(* CODESYS project UralKoksWin.project

Project tree, tasks and I/O mapping:
  Device : SPK1xx[M01], Production association OWEN, order no. 4, version 3.5.11.54
    application Application
      libraries: Standard, * (System); Util, * (System)
      task MainTask (cyclic, interval t#20ms, priority 1) calls PLC_PRG, MECH
      task VISU_TASK (cyclic, interval 100 ms, priority 31) calls VisuElems.Visu_Prg, CountWebCli
      task Task_Chain (cyclic, interval t#20ms, priority 1) calls Chain
      task TrendRecordingTask (cyclic, interval 100 ms, priority 31) calls VisuTrendStorageAccess.GlobalInstances.g_TrendRecordingManager.CyclicCall
      program PLC_PRG [LD]
      visualisation VFrADiag
      data type MV210_202
      data type MU210_402
      data type TRM201
      data type Vector75
      visualisation VFr4Baraban
      visualisation VMain
      visualisation VFr1Main
      image pool ImagePool
      visualisation VFr2KonvFrak
      visualisation VFr3Grohot
      visualisation VFr5Gorelka
      visualisation VFr6Dedusting
      text list TextList
      data type Vector100
      data type ABB330
      global variables GVL
      program MECH [CFC]
      data type PME
      data type VLT2800
      program Chain [ST]
      text list STEPS
      function block Motor [LD]
      program CountWebCli [ST]
      visualisation VFr7RandE
    Info : Info, Production association OWEN, version 3.5.11.5002
        unmapped channels: VENDOR, DEVICE, SERIAL, RUNTIME, FIRMWARE, LINUX, TARGET, PROJECT, AUTHOR, VERSION, PROFILE, LASTCHANGES
    Screen : Screen, Production association OWEN, version 3.5.11.5001
        unmapped channels: Get Brightness, Dim time, Off time, Full brightness, Dim brightness, Off brightness, Dim visu name, Off visu name, On visu name, Wake up
    Debug : Debug, Production association OWEN, version 3.5.11.5001
        unmapped channels: RAM used, RAM free, Open files, Processor usage, Core temp, Enable Debug, Debug pause
    OwenRTC : OwenRTC, Production association OWEN, version 3.5.11.5001
        unmapped channels: Year, Month, Day, Hour, Minute, Second, Day of Week, Week of Year, Format Date, Format Time, UTC Offset, NTP Enabled, NTP Error, System Timer, New Year, New Month, New Day, New Hour, New Minute, New Second, New UTC Offset, Set Settings DT, Enable NTP, Prefer Server
    OwenCloud : OwenCloud, Production association OWEN, version 3.5.11.5001
        unmapped channels: OwenCloud enabled, Enable OwenCloud, Token
    Drives : Drives, Production association OWEN, version 3.5.11.5001
        unmapped channels: FS size, FS used, FS free, USB Mounted, USB Unmount done, USB size, USB used, USB free, MMC Mounted, MMC Unmount done, MMC size, MMC used, MMC free, Enable Drives, USB Unmount, MMC Unmount
    Network : Network, Production association OWEN, version 3.5.11.5001
        unmapped channels: DHCP enabled, IP, Mask, Gateway, MAC, Hostname, Enable DHCP, New IP, New Mask, New Gateway, New Hostname, Set Settings
    Watchdog : Watchdog, Production association OWEN, version 3.5.11.5001
        unmapped channels: Exception Handling, Last Exception Code, Last Exception Description, Last Exception Time, Hardware Watchdog Flag, Reboot
    Buzzer : Buzzer, Production association OWEN, version 3.5.11.5001
        unmapped channels: Buzzer enabled, Enable Buzzer
    Ethernet : Ethernet, 3S - Smart Software Solutions GmbH, version 3.5.11.0
        settings: IPAddress = [192,168,1,151]; SubnetMask = [255,255,255,0]; GatewayAddress = [0,0,0,0]; MACAddress = [16#E4,16#1E,16#0A,16#00,16#16,16#C1]; NetworkInterfaceName = 'eth0'; NetworkInterfaceName = "eth0"; SaveCommunicationSettings = FALSE
      Modbus_TCP_Master : Modbus TCP Master, 3S - Smart Software Solutions GmbH, version 3.5.11.30
          settings: AutoReconnect = TRUE
        MU210_402DO : Modbus TCP Slave, 3S - Smart Software Solutions GmbH, version 3.5.11.30
            settings: Unit-ID = 1; IPAddress = [192, 168, 1, 153]; DO.Function Code = 16; DO.Read Offset = 0; DO.Read Length = 0; DO.Write Offset = 16#01D6; DO.Write Length = 1; DO.Cycle Time = 20
            output Application.MECH.K40.xMODBUS_Run : BOOL  // DO.DO.Bit0
            output Application.MECH.K25.xMODBUS_Run : BOOL  // DO.DO.Bit1
            output Application.MECH.K10.xMODBUS_Run : BOOL  // DO.DO.Bit2
            output Application.MECH.K0.xOUT_Run : BOOL  // DO.DO.Bit3
            output Application.MECH.Gr.xOUT_Run : BOOL  // DO.DO.Bit4
            output Application.MECH.PD.xMODBUS_Run : BOOL  // DO.DO.Bit5
            output Application.MECH.BR.xOUT_Run : BOOL  // DO.DO.Bit6
            output Application.MECH.Ded.xOUT_MODBUS_Run : BOOL  // DO.DO.Bit7
            output Application.MECH.EL.xOUT_MODBUS_Run : BOOL  // DO.DO.Bit8
            output Application.MECH.xGorRun : BOOL  // DO.DO.Bit9
            output Application.MECH.xVibRun : BOOL  // DO.DO.Bit10
            output Application.PLC_PRG.DOutput1.xDO12 : BOOL  // DO.DO.Bit11
            output Application.MECH.xGorAck : BOOL  // DO.DO.Bit12
            output Application.Chain.xLampPUSK : BOOL  // DO.DO.Bit13
            output Application.MECH.xDrob_OUT_Run : BOOL  // DO.DO.Bit14
            output Application.PLC_PRG.DOutput1.xDO16 : BOOL  // DO.DO.Bit15
            unmapped channels: DO
        MV210_202DI : Modbus TCP Slave, 3S - Smart Software Solutions GmbH, version 3.5.11.30
            settings: Unit-ID = 1; IPAddress = [192, 168, 1, 152]; DI.Function Code = 3; DI.Read Offset = 16#0033; DI.Read Length = 2; DI.Write Offset = 0; DI.Write Length = 0; DI.Cycle Time = 20
            input  Application.PLC_PRG.DInput1.xDI1 : BOOL  // DI.DI.Bit0
            input  Application.PLC_PRG.DInput1.xDI2 : BOOL  // DI.DI.Bit1
            input  Application.PLC_PRG.DInput1.xDI3 : BOOL  // DI.DI.Bit2
            input  Application.PLC_PRG.DInput1.xDI4 : BOOL  // DI.DI.Bit3
            input  Application.PLC_PRG.DInput1.xDI5 : BOOL  // DI.DI.Bit4
            input  Application.PLC_PRG.DInput1.xDI6 : BOOL  // DI.DI.Bit5
            input  Application.PLC_PRG.DInput1.xDI7 : BOOL  // DI.DI.Bit6
            input  Application.PLC_PRG.DInput1.xDI8 : BOOL  // DI.DI.Bit7
            input  Application.PLC_PRG.DInput1.xDI9 : BOOL  // DI.DI.Bit8
            input  Application.PLC_PRG.DInput1.xDI10 : BOOL  // DI.DI.Bit9
            input  Application.PLC_PRG.DInput1.xDI11 : BOOL  // DI.DI.Bit10
            input  Application.PLC_PRG.DInput1.xDI12 : BOOL  // DI.DI.Bit11
            input  Application.PLC_PRG.DInput1.xDI13 : BOOL  // DI.DI.Bit12
            input  Application.PLC_PRG.DInput1.xDI14 : BOOL  // DI.DI.Bit13
            input  Application.PLC_PRG.DInput1.xDI15 : BOOL  // DI.DI.Bit14
            input  Application.PLC_PRG.DInput1.xDI16 : BOOL  // DI.DI.Bit15
            input  Application.PLC_PRG.DInput1.xDI17 : BOOL  // DI.DI.Bit0
            input  Application.PLC_PRG.DInput1.xDI18 : BOOL  // DI.DI.Bit1
            input  Application.PLC_PRG.DInput1.xDI19 : BOOL  // DI.DI.Bit2
            input  Application.PLC_PRG.DInput1.xDI20 : BOOL  // DI.DI.Bit3
            unmapped channels: DI
        MV210_202DI2 : Modbus TCP Slave, 3S - Smart Software Solutions GmbH, version 3.5.11.30
            settings: Unit-ID = 1; IPAddress = [192, 168, 1, 154]; DI.Function Code = 3; DI.Read Offset = 16#0033; DI.Read Length = 2; DI.Write Offset = 0; DI.Write Length = 0; DI.Cycle Time = 20
            input  Application.PLC_PRG.DInput2.xDI1 : BOOL  // DI.DI.Bit0
            input  Application.PLC_PRG.DInput2.xDI2 : BOOL  // DI.DI.Bit1
            input  Application.MECH.xGorFault : BOOL  // DI.DI.Bit2
            input  Application.MECH.xGorWork : BOOL  // DI.DI.Bit3
            input  Application.MECH.xGor2Stup : BOOL  // DI.DI.Bit4
            input  Application.PLC_PRG.DInput2.xDI6 : BOOL  // DI.DI.Bit5
            input  Application.PLC_PRG.DInput2.xDI7 : BOOL  // DI.DI.Bit6
            input  Application.PLC_PRG.DInput2.xDI8 : BOOL  // DI.DI.Bit7
            input  Application.PLC_PRG.DInput2.xDI9 : BOOL  // DI.DI.Bit8
            input  Application.PLC_PRG.DInput2.xDI10 : BOOL  // DI.DI.Bit9
            input  Application.PLC_PRG.DInput2.xDI11 : BOOL  // DI.DI.Bit10
            input  Application.PLC_PRG.DInput2.xDI12 : BOOL  // DI.DI.Bit11
            input  Application.PLC_PRG.DInput2.xDI13 : BOOL  // DI.DI.Bit12
            input  Application.PLC_PRG.DInput2.xDI14 : BOOL  // DI.DI.Bit13
            input  Application.PLC_PRG.DInput2.xDI15 : BOOL  // DI.DI.Bit14
            input  Application.PLC_PRG.DInput2.xDI16 : BOOL  // DI.DI.Bit15
            input  Application.PLC_PRG.DInput2.xDI17 : BOOL  // DI.DI.Bit0
            input  Application.PLC_PRG.DInput2.xDI18 : BOOL  // DI.DI.Bit1
            input  Application.PLC_PRG.DInput2.xDI19 : BOOL  // DI.DI.Bit2
            input  Application.PLC_PRG.DInput2.xDI20 : BOOL  // DI.DI.Bit3
            unmapped channels: DI
    COM2 : Modbus COM, 3S - Smart Software Solutions GmbH, version 3.5.11.20
        settings: DataBits = 8; StopBits = 2; ComPort = 2
      Master_2 : Modbus Master, COM Port, 3S - Smart Software Solutions GmbH, version 3.5.11.20
          settings: Transmission = 'RTU'; ResponseTimeout = 1000; TimeBetweenFrames = 20; Auto-restart communication = TRUE
        DedustingSlave : Modbus Slave, COM Port, 3S - Smart Software Solutions GmbH, version 3.5.10.30
            settings: SlaveAddress = 30; ResponseTimeout = 1000; UseExtendedFunctionCodes = TRUE; Current.Function Code = 3; Current.Read Offset = 16#1004; Current.Read Length = 1; Current.Write Offset = 0; Current.Write Length = 0; Current.Cycle Time = 1000; PVSpeed.Function Code = 3; PVSpeed.Read Offset = 16#1001; PVSpeed.Read Length = 1; PVSpeed.Write Offset = 0; PVSpeed.Write Length = 0; PVSpeed.Cycle Time = 1000; SPSpeed.Function Code = 6; SPSpeed.Read Offset = 0; SPSpeed.Read Length = 0; SPSpeed.Write Offset = 16#1000; SPSpeed.Write Length = 1; SPSpeed.Cycle Time = 1000
            input  Application.MECH.Ded.iIN_MODBUS_Iengie : WORD  // Current.Current
            input  Application.MECH.Ded.iIN_MODBUS_PVSpeed : WORD  // PVSpeed.PVSpeed
            output Application.MECH.Ded.iOUT_MODBUS_SPSpeed : WORD  // SPSpeed.SPSpeed
            unmapped channels: Current, PVSpeed, SPSpeed
        ElevatorSlave : Modbus Slave, COM Port, 3S - Smart Software Solutions GmbH, version 3.5.10.30
            settings: SlaveAddress = 25; ResponseTimeout = 1000; UseExtendedFunctionCodes = TRUE; PVSpeed.Function Code = 3; PVSpeed.Read Offset = 16#1001; PVSpeed.Read Length = 1; PVSpeed.Write Offset = 0; PVSpeed.Write Length = 0; PVSpeed.Cycle Time = 1000; Current.Function Code = 3; Current.Read Offset = 16#1004; Current.Read Length = 1; Current.Write Offset = 0; Current.Write Length = 0; Current.Cycle Time = 1000; SPspeed.Function Code = 6; SPspeed.Read Offset = 0; SPspeed.Read Length = 0; SPspeed.Write Offset = 16#1000; SPspeed.Write Length = 1; SPspeed.Cycle Time = 1000
            input  Application.MECH.EL.iIN_MODBUS_PVSpeed : WORD  // PVSpeed.PVSpeed
            input  Application.MECH.EL.iIN_MODBUS_Iengie : WORD  // Current.Current
            output Application.MECH.EL.iOUT_MODBUS_SPSpeed : WORD  // SPspeed.SPspeed
            unmapped channels: PVSpeed, Current, SPspeed
        VentilatorSlave : Modbus Slave, COM Port, 3S - Smart Software Solutions GmbH, version 3.5.10.30
            settings: SlaveAddress = 35; ResponseTimeout = 1000; UseExtendedFunctionCodes = TRUE; PVSpeed.Function Code = 3; PVSpeed.Read Offset = 16#1001; PVSpeed.Read Length = 1; PVSpeed.Write Offset = 0; PVSpeed.Write Length = 0; PVSpeed.Cycle Time = 1000; StatWord.Function Code = 3; StatWord.Read Offset = 16#3000; StatWord.Read Length = 1; StatWord.Write Offset = 0; StatWord.Write Length = 0; StatWord.Cycle Time = 1000; BR_Speed.Function Code = 3; BR_Speed.Read Offset = 16#100B; BR_Speed.Read Length = 1; BR_Speed.Write Offset = 0; BR_Speed.Write Length = 0; BR_Speed.Cycle Time = 100
            input  Application.MECH.iInMBVentPVSpeed : WORD  // PVSpeed.PVSpeed
            input  Application.MECH.xVentWorkBit1 : BOOL  // StatWord.StatWord.Bit0
            input  Application.MECH.xVentWorkBit2 : BOOL  // StatWord.StatWord.Bit1
            input  Application.MECH.BR.iIN_MODBUS_PVSpeed : WORD  // BR_Speed.BR_Speed
            unmapped channels: PVSpeed, StatWord, BR_Speed
    COM1 : Modbus COM, 3S - Smart Software Solutions GmbH, version 3.5.11.20
        settings: DataBits = 8; StopBits = 2; ComPort = 1
      Master_1 : Modbus Master, COM Port, 3S - Smart Software Solutions GmbH, version 3.5.11.20
          settings: Transmission = 'RTU'; ResponseTimeout = 1000; TimeBetweenFrames = 10; Auto-restart communication = TRUE
        Konv40Slave : Modbus Slave, COM Port, 3S - Smart Software Solutions GmbH, version 3.5.10.30
            settings: SlaveAddress = 5; ResponseTimeout = 1000; UseExtendedFunctionCodes = TRUE; SPSpeed.Function Code = 6; SPSpeed.Read Offset = 0; SPSpeed.Read Length = 0; SPSpeed.Write Offset = 16#1000; SPSpeed.Write Length = 1; SPSpeed.Cycle Time = 1000; PVSpeed.Function Code = 3; PVSpeed.Read Offset = 16#1001; PVSpeed.Read Length = 1; PVSpeed.Write Offset = 0; PVSpeed.Write Length = 0; PVSpeed.Cycle Time = 1000; Current.Function Code = 3; Current.Read Offset = 16#1004; Current.Read Length = 1; Current.Write Offset = 0; Current.Write Length = 0; Current.Cycle Time = 1000; MI.Function Code = 3; MI.Read Offset = 16#1008; MI.Read Length = 1; MI.Write Offset = 0; MI.Write Length = 0; MI.Cycle Time = 1000
            output Application.MECH.K40.iMODBUS_SPSpeed : WORD  // SPSpeed.SPSpeed
            input  Application.MECH.K40.iMODBUS_PVSpeed : WORD  // PVSpeed.PVSpeed
            input  Application.MECH.K40.iMODBUS_Iengie : WORD  // Current.Current
            input  Application.MECH.KM_K0 : BOOL  // MI.MI.Bit3
            input  Application.MECH.KM_Gr : BOOL  // MI.MI.Bit4
            unmapped channels: SPSpeed, PVSpeed, Current, MI
        PodachaSlave : Modbus Slave, COM Port, 3S - Smart Software Solutions GmbH, version 3.5.10.30
            settings: SlaveAddress = 20; ResponseTimeout = 1000; UseExtendedFunctionCodes = TRUE; PVSpeed.Function Code = 3; PVSpeed.Read Offset = 16#0004; PVSpeed.Read Length = 3; PVSpeed.Write Offset = 0; PVSpeed.Write Length = 0; PVSpeed.Cycle Time = 1000
            input  Application.MECH.PD.iMODBUS_SPSpeed : WORD  // PVSpeed.PVSpeed
            input  Application.MECH.PD.iMODBUS_PVSpeed : WORD  // PVSpeed.PVSpeed
            input  Application.MECH.PD.iMODBUS_Iengie : WORD  // PVSpeed.PVSpeed
            unmapped channels: PVSpeed
        Konv25Slave : Modbus Slave, COM Port, 3S - Smart Software Solutions GmbH, version 3.5.10.30
            settings: SlaveAddress = 10; ResponseTimeout = 1000; UseExtendedFunctionCodes = TRUE; SPSpeed.Function Code = 6; SPSpeed.Read Offset = 0; SPSpeed.Read Length = 0; SPSpeed.Write Offset = 16#1000; SPSpeed.Write Length = 1; SPSpeed.Cycle Time = 1000; PVSpeed.Function Code = 3; PVSpeed.Read Offset = 16#1001; PVSpeed.Read Length = 1; PVSpeed.Write Offset = 0; PVSpeed.Write Length = 0; PVSpeed.Cycle Time = 1000; Current.Function Code = 3; Current.Read Offset = 16#1004; Current.Read Length = 1; Current.Write Offset = 0; Current.Write Length = 0; Current.Cycle Time = 1000
            output Application.MECH.K25.iMODBUS_SPSpeed : WORD  // SPSpeed.SPSpeed
            input  Application.MECH.K25.iMODBUS_PVSpeed : WORD  // PVSpeed.PVSpeed
            input  Application.MECH.K25.iMODBUS_Iengie : WORD  // Current.Current
            unmapped channels: SPSpeed, PVSpeed, Current
        Konv10Slave : Modbus Slave, COM Port, 3S - Smart Software Solutions GmbH, version 3.5.10.30
            settings: SlaveAddress = 15; ResponseTimeout = 1000; UseExtendedFunctionCodes = TRUE; SPSpeed.Function Code = 6; SPSpeed.Read Offset = 0; SPSpeed.Read Length = 0; SPSpeed.Write Offset = 16#1000; SPSpeed.Write Length = 1; SPSpeed.Cycle Time = 1000; PVSpeed.Function Code = 3; PVSpeed.Read Offset = 16#1001; PVSpeed.Read Length = 1; PVSpeed.Write Offset = 0; PVSpeed.Write Length = 0; PVSpeed.Cycle Time = 1000; Current.Function Code = 3; Current.Read Offset = 16#1004; Current.Read Length = 1; Current.Write Offset = 0; Current.Write Length = 0; Current.Cycle Time = 1000
            output Application.MECH.K10.iMODBUS_SPSpeed : WORD  // SPSpeed.SPSpeed
            input  Application.MECH.K10.iMODBUS_PVSpeed : WORD  // PVSpeed.PVSpeed
            input  Application.MECH.K10.iMODBUS_Iengie : WORD  // Current.Current
            unmapped channels: SPSpeed, PVSpeed, Current
    COM3 : Modbus COM, 3S - Smart Software Solutions GmbH, version 3.5.11.20
        settings: DataBits = 8; StopBits = 2; ComPort = 3
      Master_3 : Modbus Master, COM Port, 3S - Smart Software Solutions GmbH, version 3.5.11.20
          settings: Transmission = 'RTU'; ResponseTimeout = 1000; TimeBetweenFrames = 10; Auto-restart communication = TRUE
        TRMGorelkaSlave : Modbus Slave, COM Port, 3S - Smart Software Solutions GmbH, version 3.5.10.30
            settings: SlaveAddress = 40; ResponseTimeout = 1000; UseExtendedFunctionCodes = TRUE; PV_SP.Function Code = 3; PV_SP.Read Offset = 16#0001; PV_SP.Read Length = 1; PV_SP.Write Offset = 0; PV_SP.Write Length = 0; PV_SP.Cycle Time = 1000; temp_SP.Function Code = 3; temp_SP.Read Offset = 16#0002; temp_SP.Read Length = 1; temp_SP.Write Offset = 0; temp_SP.Write Length = 0; temp_SP.Cycle Time = 1000; STAT.Function Code = 3; STAT.Read Offset = 16#0000; STAT.Read Length = 1; STAT.Write Offset = 0; STAT.Write Length = 0; STAT.Cycle Time = 1000
            input  Application.MECH.iInMBGorPVTemp : WORD  // PV_SP.PV_SP
            input  Application.MECH.iInMBGorSPTemp : WORD  // temp_SP.temp_SP
            input  Application.MECH.xGorNagrevONOFF : BOOL  // STAT.STAT.Bit4
            unmapped channels: PV_SP, temp_SP, STAT
        TRMDedustingSlave : Modbus Slave, COM Port, 3S - Smart Software Solutions GmbH, version 3.5.10.30
            settings: SlaveAddress = 45; ResponseTimeout = 1000; UseExtendedFunctionCodes = TRUE; PV_SP.Function Code = 3; PV_SP.Read Offset = 16#0001; PV_SP.Read Length = 1; PV_SP.Write Offset = 0; PV_SP.Write Length = 0; PV_SP.Cycle Time = 1000
            input  Application.MECH.iInMBDedPVTemp : WORD  // PV_SP.PV_SP
            unmapped channels: PV_SP
  text list GlobalTextList
  5ce3da45-db07-42e7-a21c-a00fff4ed8f6|img\fonFrame.png
  text list System
  5ce3da45-db07-42e7-a21c-a00fff4ed8f6|img\frame1.png
  5ce3da45-db07-42e7-a21c-a00fff4ed8f6|img\333.png
*)

// Device/Application/MV210_202
TYPE MV210_202 :
STRUCT
	xDI1: BOOL;
	xDI2: BOOL;
	xDI3: BOOL;
	xDI4: BOOL;
	xDI5: BOOL;
	xDI6: BOOL;
	xDI7: BOOL;
	xDI8: BOOL;
	xDI9: BOOL;
	xDI10: BOOL;
	xDI11: BOOL;
	xDI12: BOOL;
	xDI13: BOOL;
	xDI14: BOOL;
	xDI15: BOOL;
	xDI16: BOOL;
	xDI17: BOOL;
	xDI18: BOOL;
	xDI19: BOOL;
	xDI20: BOOL;
END_STRUCT
END_TYPE

// Device/Application/MU210_402
TYPE MU210_402 :
STRUCT
	xDO1: BOOL;
	xDO2: BOOL;
	xDO3: BOOL;
	xDO4: BOOL;
	xDO5: BOOL;
	xDO6: BOOL;
	xDO7: BOOL;
	xDO8: BOOL;
	xDO9: BOOL;
	xDO10: BOOL;
	xDO11: BOOL;
	xDO12: BOOL;
	xDO13: BOOL;
	xDO14: BOOL;
	xDO15: BOOL;
	xDO16: BOOL;
END_STRUCT
END_TYPE

// Device/Application/TRM201
TYPE TRM201 :
STRUCT
	iPV: INT;
	iSP: INT;
	nagrevONOFF: BOOL;
	
END_STRUCT
END_TYPE

// Device/Application/Vector75
TYPE Vector75 :
STRUCT
	iOUT_MODBUS_SPSpeed,
	iIN_MODBUS_PVSpeed,
	iIN_MODBUS_Iengie: INT;
	

	xIN_Run: BOOL;
	xOUT_MODBUS_Run:BOOL;
	xOUT_Ready: BOOL;
	xOUT_Error: BOOL;
	xOUT_Work: BOOL;

	xIN_Error: BOOL;

	iOUT_PVRotation: INT;
	iOUT_PVSpeed: INT; 

	rOUT_Current: REAL;
	
	iIN_MODBUS_AI: INT;
END_STRUCT
END_TYPE

// Device/Application/Vector100
TYPE Vector100 :
STRUCT
	iMODBUS_SPSpeed,
	iMODBUS_PVSpeed,
	iMODBUS_Iengie: INT;
	

	xIN_Run: BOOL;
	xMODBUS_Run:BOOL;
	xOUT_Ready: BOOL;
	xOUT_Error: BOOL;
	xOUT_Work: BOOL;

	xIN_Error: BOOL;

	iOUT_PVRotation: INT;
	iOUT_PVSpeed: INT; 

	rOUT_Current: REAL;
	
END_STRUCT
END_TYPE

// Device/Application/ABB330
TYPE ABB330 :
STRUCT
	iMODBUS_SPSpeed,
	iMODBUS_PVSpeed,
	iMODBUS_Iengie: INT;
	

	xIN_Run: BOOL;
	xMODBUS_Run:BOOL;
	xOUT_Ready: BOOL;
	xOUT_Error: BOOL;
	xOUT_Work: BOOL;

	xIN_Error: BOOL;

	iOUT_PVRotation: INT;
	iOUT_PVSpeed: INT; 

	rOUT_Current: REAL;
	
END_STRUCT
END_TYPE

// Device/Application/PME
TYPE PME :
STRUCT

	xIN_Run: BOOL;
	xIN_Error: BOOL;

	
	
	xOUT_Ready: BOOL;
	xOUT_Error: BOOL;
	xOUT_Work: BOOL;
	xOUT_Run: BOOL;
	
	iOUT_PVSpeed: INT;
	

	iOUT_PVRotation: INT;
	
END_STRUCT
END_TYPE

// Device/Application/VLT2800
TYPE VLT2800 :
STRUCT
	xIN_Run: BOOL;
	xIN_Error: BOOL;
	
	xOUT_Ready: BOOL;
	xOUT_Error: BOOL;
	xOUT_Work: BOOL;
	xOUT_Run: BOOL;
	
	iIN_MODBUS_PVSpeed: INT;
	rOUT_PVSpeed: REAL;
END_STRUCT
END_TYPE

// Device/Application/GVL
{attribute 'qualified_only'}
VAR_GLOBAL

END_VAR

// Device/Application/PLC_PRG
PROGRAM PLC_PRG
VAR

	xAck :BOOL;
	DInput1: MV210_202;
	DInput2: MV210_202;
	DOutput1: MU210_402;
	xFlash: BOOL;
	Flasing: BLINK;
END_VAR

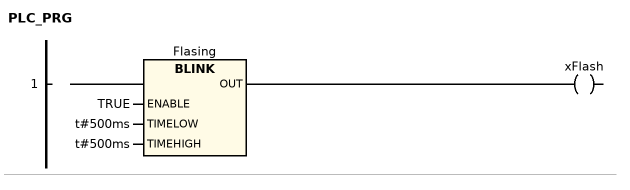
// NETWORK 1
Flasing(ENABLE := TRUE, TIMELOW := t#500ms, TIMEHIGH := t#500ms); // BLINK
xFlash := Flasing.OUT;

END_PROGRAM

// Device/Application/MECH
PROGRAM MECH
VAR
	Konveer40: Motor;
	Konveer25: Motor;
	Konveer10: Motor;
	Konveer0: Motor;
	Grohot: Motor;
	Podacha: Motor;
	Baraban: Motor;
	Elevator: Motor;
	Dedusting: Motor;
	Drobilka: Motor;
	
	xVibRun,  xVibTEST : BOOL;
	VIBRATOR: BLINK;
	iSP_Podacha: INT;
	xVentWorkBit1: BOOL;
	xVentWorkBit2: BOOL;
	xVentWork: BOOL;
	iInMBVentPVSpeed: INT;
	rOutVentPVSpeed: REAL;
	
	xGorFault: BOOL;
	xGorWork:BOOL;
	xGor2Stup:BOOL;
	xGorOprob:BOOL;
	xGorRun:BOOL;
	xGorNagrevONOFF:BOOL;
	xGorAckButton:BOOL;
	
	iInMBGorPVTemp: INT;
	iInMBGorSPTemp: INT;
	iInMBDedPVTemp: INT;
	rOutGorPVTemp: LREAL;
	rOutGorSPTemp: LREAL;
	rOutDedPVTemp: LREAL;
	KM_K0: BOOL;
	KM_Gr: BOOL;
	xGorFaultRS: RS;
	xGorAck: BOOL;
	AckGor: TOF;
	
	
	xDrob_OUT_Work: BOOL;
	xDrob_OUT_Error: BOOL;
	xDrob_OUT_Ready: BOOL;
	xDrob_OUT_Run: BOOL;
END_VAR

VAR_INPUT
	K40:Vector100;
	K25:Vector100;
	K10:Vector100;
	K0: PME;
	Gr: PME;
	PD: ABB330;
	BR: VLT2800;
	EL: Vector75;
	Ded: Vector75;
	xVibRunAUTO: BOOL;
	xGorRunAUTO: BOOL;
	xDrobRun: BOOL;
END_VAR

VAR RETAIN
	iVibWork: INT:=2;
	iVibPause: INT:=30;
	xVibEnable: BOOL:=FALSE;
	
	K40_iIN_SPSpeed: INT:=20;
	K40_xIN_EnCtrlSensor: BOOL:=TRUE;
	K40_iIN_SPRotatTimeMS: INT:=6300;
	
	K25_iIN_SPSpeed: INT:=25;
	K25_xIN_EnCtrlSensor: BOOL:=TRUE;
	K25_iIN_SPRotatTimeMS: INT:=4000;
	
	K10_xIN_EnCtrlSensor: BOOL:=TRUE;
	K10_iIN_SPSpeed: INT:=30;
	K10_iIN_SPRotatTimeMS: INT:=3000;
	
	K0_xIN_EnCtrlSensor: BOOL:=TRUE;
	K0_iIN_SPRotatTimeMS: INT:=3000;
	
	PD_iIN_SPSpeed: INT:=27;
	PD_xIN_EnCtrlSensor: BOOL:=TRUE;
	PD_iIN_SPRotatTimeMS: INT:=3000;
	
	EL_iIN_SPSpeed: INT:=60;
	EL_xIN_EnCtrlSensor: BOOL:=TRUE;
	EL_iIN_SPRotatTimeMS: INT:=8000;
	
	Ded_iIN_SPSpeed: INT:=45;
	
	xGorSwitchRun:BOOL;
END_VAR

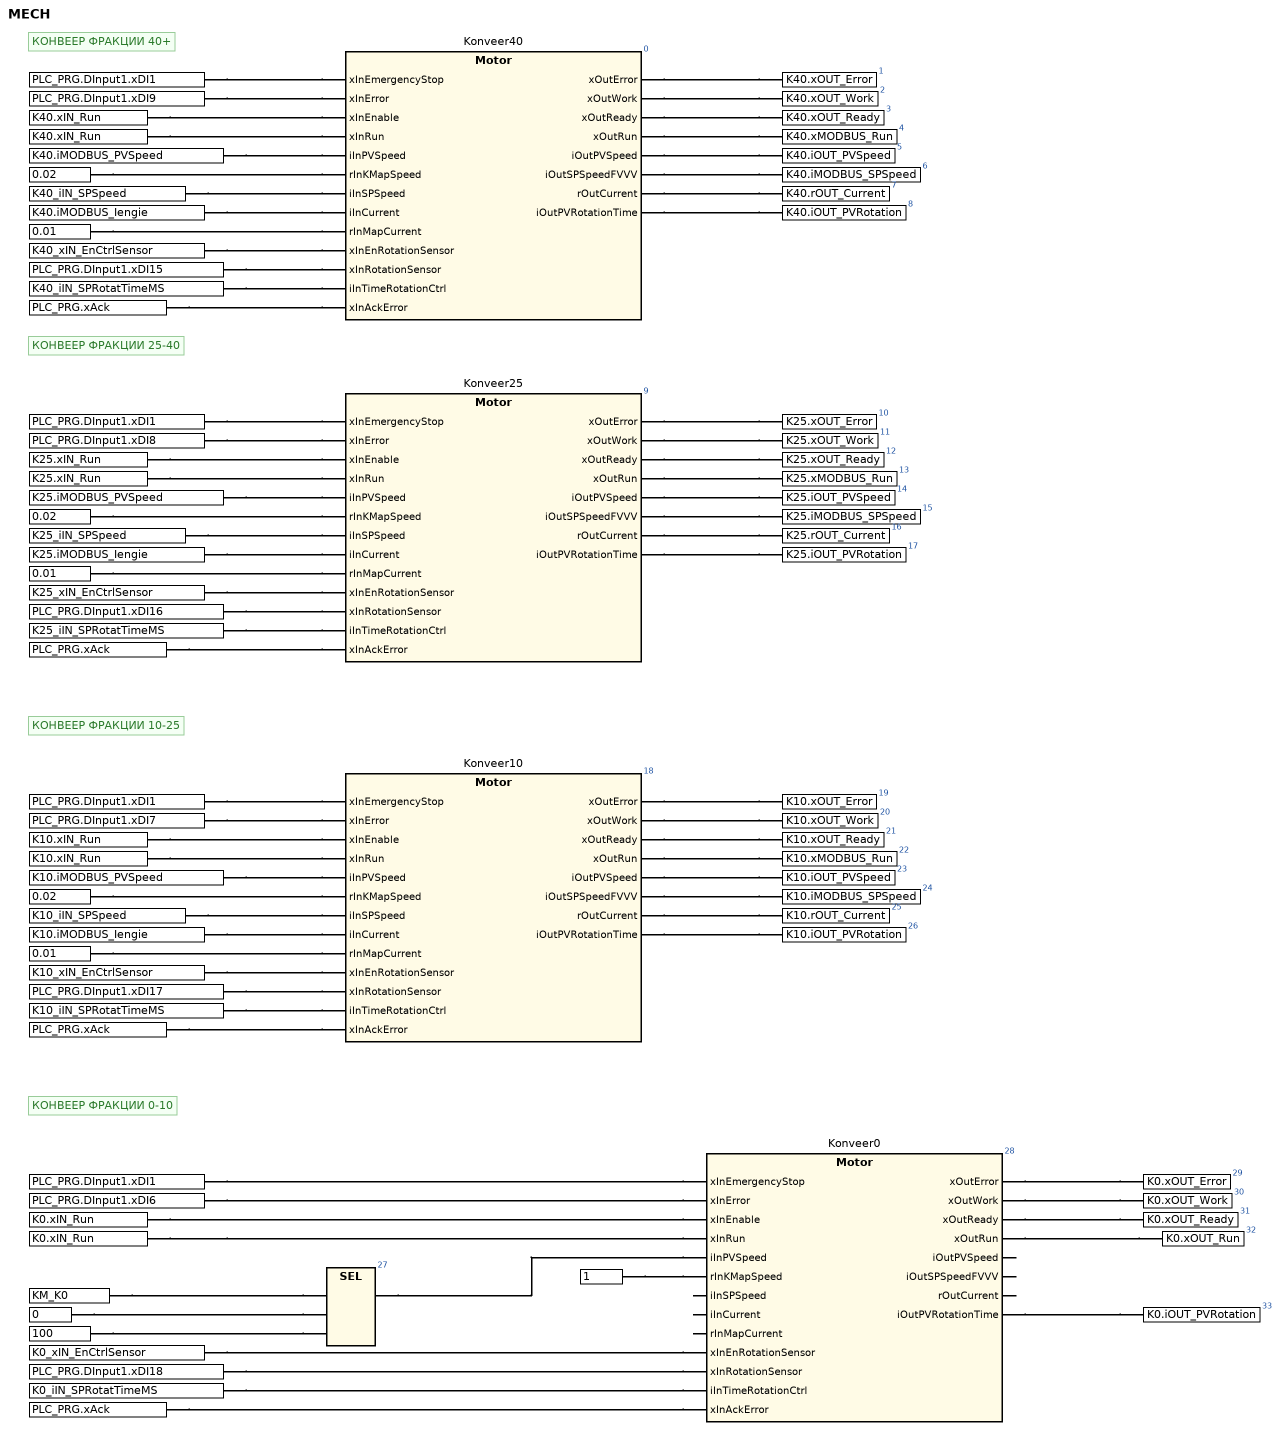
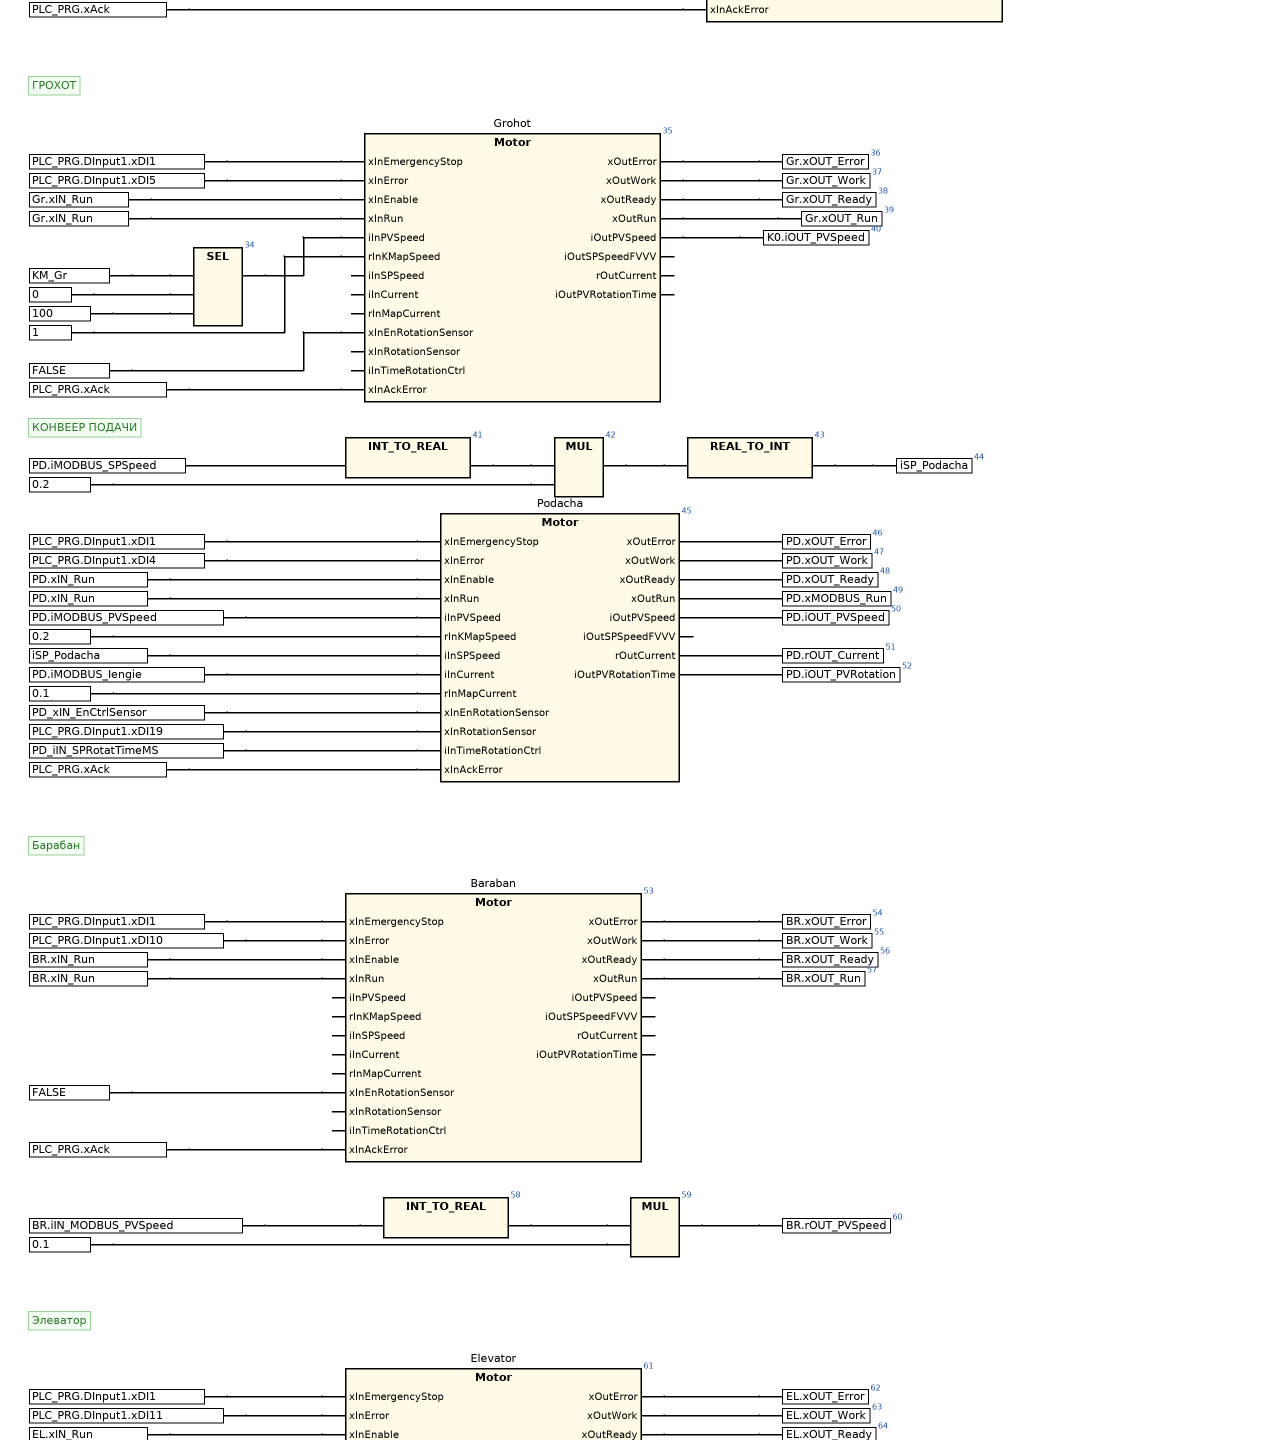
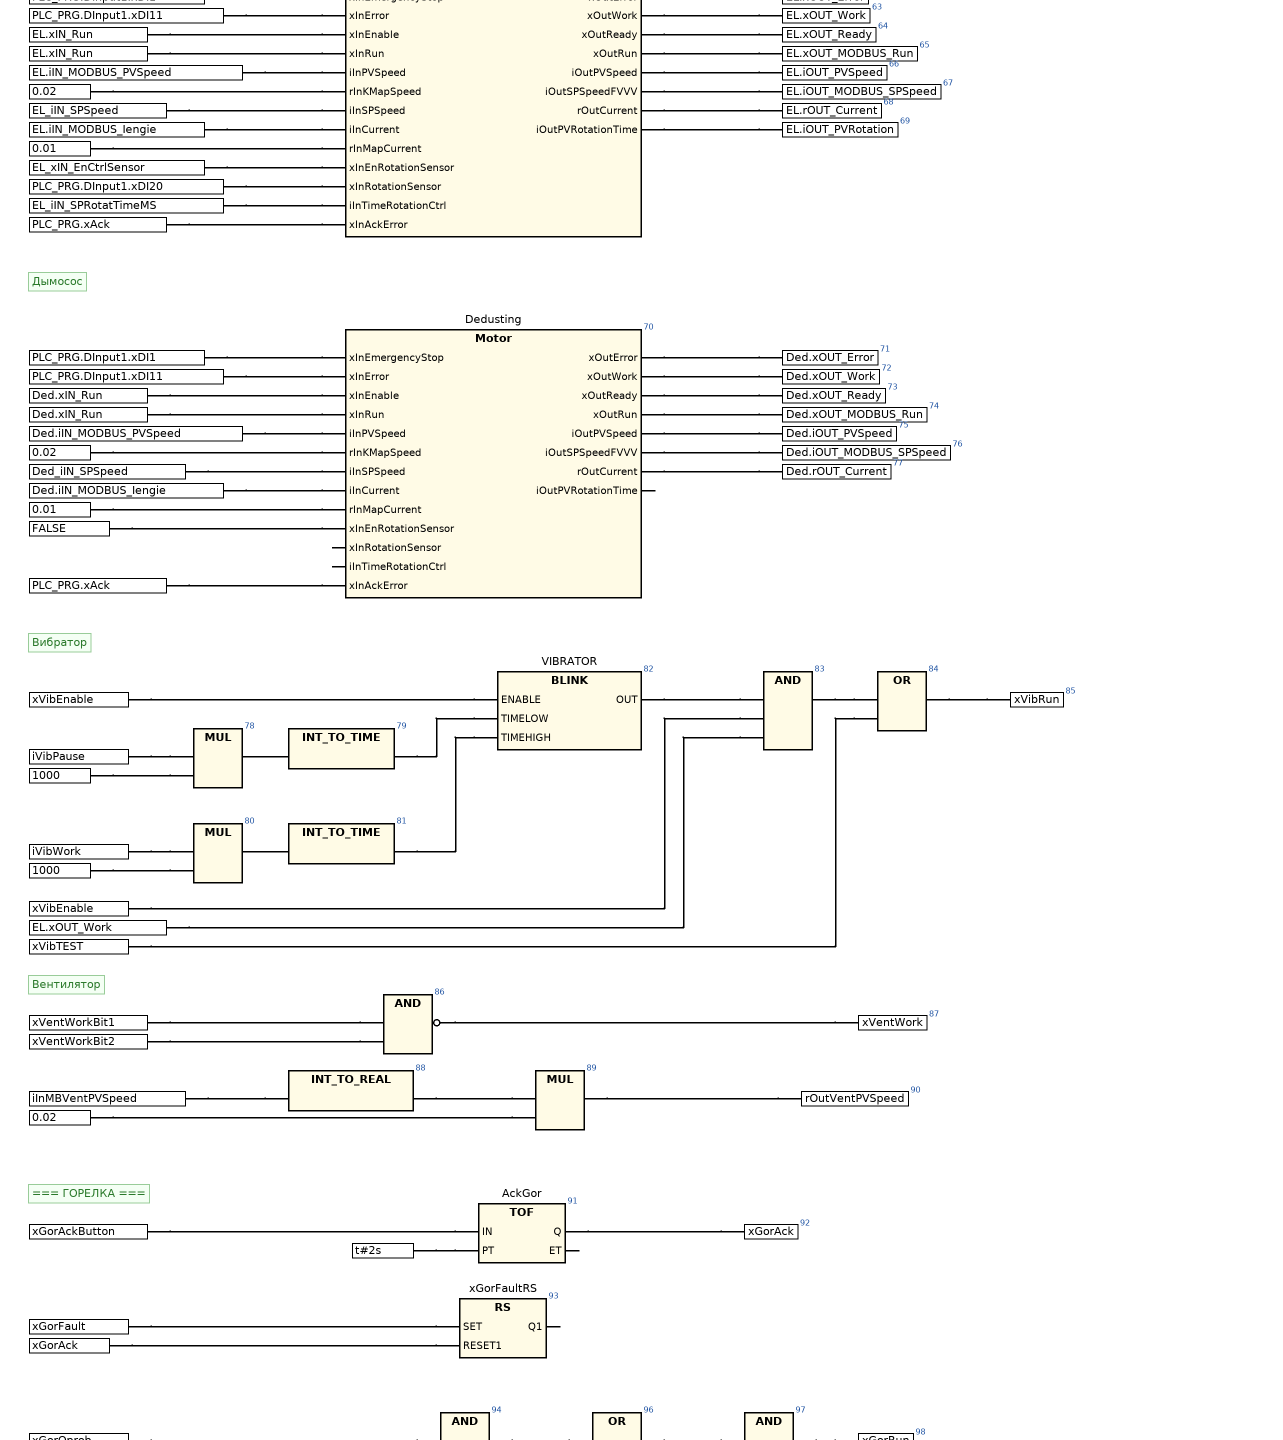
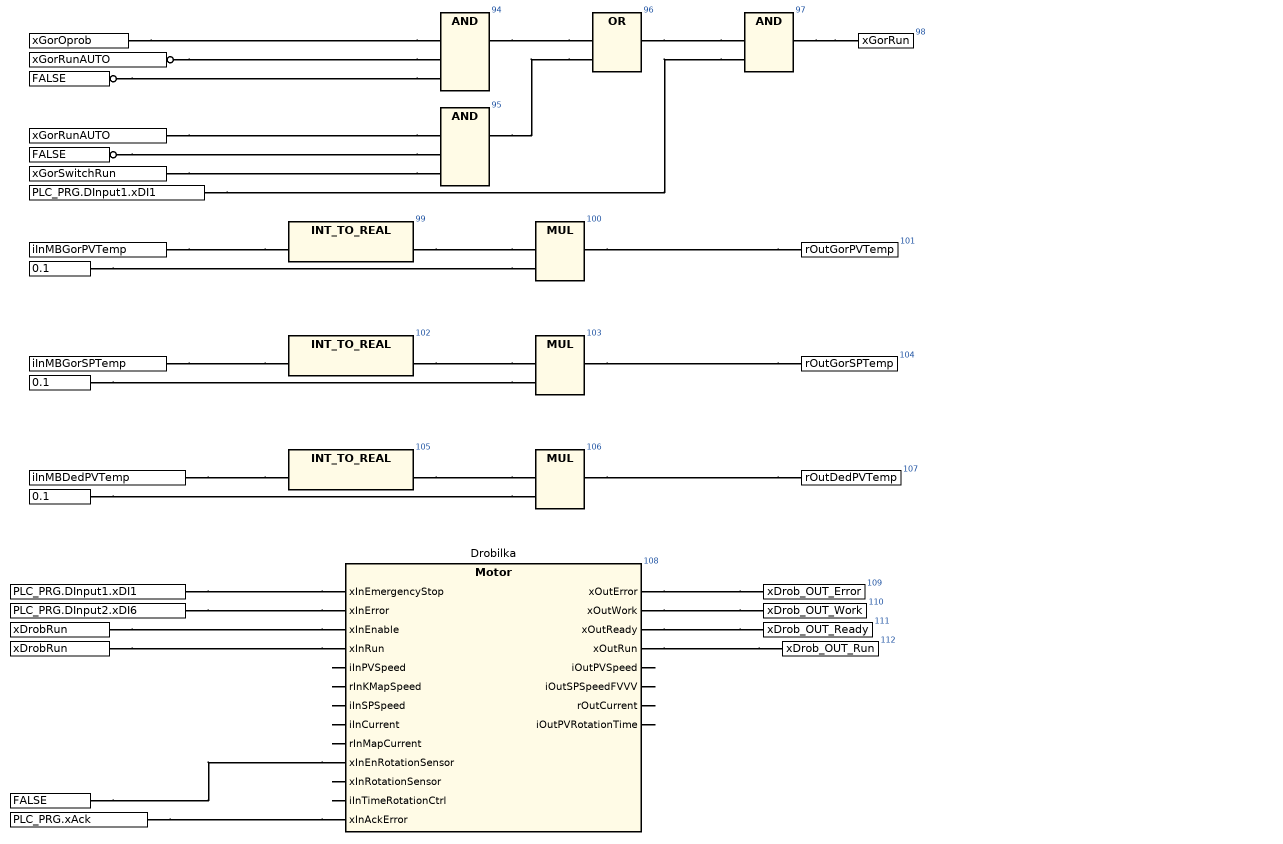
// КОНВЕЕР ФРАКЦИИ 40+
Konveer40(
    xInEmergencyStop := PLC_PRG.DInput1.xDI1,
    xInError := PLC_PRG.DInput1.xDI9,
    xInEnable := K40.xIN_Run,
    xInRun := K40.xIN_Run,
    iInPVSpeed := K40.iMODBUS_PVSpeed,
    rInKMapSpeed := 0.02,
    iInSPSpeed := K40_iIN_SPSpeed,
    iInCurrent := K40.iMODBUS_Iengie,
    rInMapCurrent := 0.01,
    xInEnRotationSensor := K40_xIN_EnCtrlSensor,
    xInRotationSensor := PLC_PRG.DInput1.xDI15,
    iInTimeRotationCtrl := K40_iIN_SPRotatTimeMS,
    xInAckError := PLC_PRG.xAck); // Motor
K40.xOUT_Error := Konveer40.xOutError;
K40.xOUT_Work := Konveer40.xOutWork;
K40.xOUT_Ready := Konveer40.xOutReady;
K40.xMODBUS_Run := Konveer40.xOutRun;
K40.iOUT_PVSpeed := Konveer40.iOutPVSpeed;
K40.iMODBUS_SPSpeed := Konveer40.iOutSPSpeedFVVV;
K40.rOUT_Current := Konveer40.rOutCurrent;
K40.iOUT_PVRotation := Konveer40.iOutPVRotationTime;
// КОНВЕЕР ФРАКЦИИ 25-40
Konveer25(
    xInEmergencyStop := PLC_PRG.DInput1.xDI1,
    xInError := PLC_PRG.DInput1.xDI8,
    xInEnable := K25.xIN_Run,
    xInRun := K25.xIN_Run,
    iInPVSpeed := K25.iMODBUS_PVSpeed,
    rInKMapSpeed := 0.02,
    iInSPSpeed := K25_iIN_SPSpeed,
    iInCurrent := K25.iMODBUS_Iengie,
    rInMapCurrent := 0.01,
    xInEnRotationSensor := K25_xIN_EnCtrlSensor,
    xInRotationSensor := PLC_PRG.DInput1.xDI16,
    iInTimeRotationCtrl := K25_iIN_SPRotatTimeMS,
    xInAckError := PLC_PRG.xAck); // Motor
K25.xOUT_Error := Konveer25.xOutError;
K25.xOUT_Work := Konveer25.xOutWork;
K25.xOUT_Ready := Konveer25.xOutReady;
K25.xMODBUS_Run := Konveer25.xOutRun;
K25.iOUT_PVSpeed := Konveer25.iOutPVSpeed;
K25.iMODBUS_SPSpeed := Konveer25.iOutSPSpeedFVVV;
K25.rOUT_Current := Konveer25.rOutCurrent;
K25.iOUT_PVRotation := Konveer25.iOutPVRotationTime;
// КОНВЕЕР ФРАКЦИИ 10-25
Konveer10(
    xInEmergencyStop := PLC_PRG.DInput1.xDI1,
    xInError := PLC_PRG.DInput1.xDI7,
    xInEnable := K10.xIN_Run,
    xInRun := K10.xIN_Run,
    iInPVSpeed := K10.iMODBUS_PVSpeed,
    rInKMapSpeed := 0.02,
    iInSPSpeed := K10_iIN_SPSpeed,
    iInCurrent := K10.iMODBUS_Iengie,
    rInMapCurrent := 0.01,
    xInEnRotationSensor := K10_xIN_EnCtrlSensor,
    xInRotationSensor := PLC_PRG.DInput1.xDI17,
    iInTimeRotationCtrl := K10_iIN_SPRotatTimeMS,
    xInAckError := PLC_PRG.xAck); // Motor
K10.xOUT_Error := Konveer10.xOutError;
K10.xOUT_Work := Konveer10.xOutWork;
K10.xOUT_Ready := Konveer10.xOutReady;
K10.xMODBUS_Run := Konveer10.xOutRun;
K10.iOUT_PVSpeed := Konveer10.iOutPVSpeed;
K10.iMODBUS_SPSpeed := Konveer10.iOutSPSpeedFVVV;
K10.rOUT_Current := Konveer10.rOutCurrent;
K10.iOUT_PVRotation := Konveer10.iOutPVRotationTime;
// КОНВЕЕР ФРАКЦИИ 0-10
Konveer0(
    xInEmergencyStop := PLC_PRG.DInput1.xDI1,
    xInError := PLC_PRG.DInput1.xDI6,
    xInEnable := K0.xIN_Run,
    xInRun := K0.xIN_Run,
    iInPVSpeed := SEL(KM_K0, 0, 100),
    rInKMapSpeed := 1,
    xInEnRotationSensor := K0_xIN_EnCtrlSensor,
    xInRotationSensor := PLC_PRG.DInput1.xDI18,
    iInTimeRotationCtrl := K0_iIN_SPRotatTimeMS,
    xInAckError := PLC_PRG.xAck); // Motor
K0.xOUT_Error := Konveer0.xOutError;
K0.xOUT_Work := Konveer0.xOutWork;
K0.xOUT_Ready := Konveer0.xOutReady;
K0.xOUT_Run := Konveer0.xOutRun;
K0.iOUT_PVRotation := Konveer0.iOutPVRotationTime;
// ГРОХОТ
Grohot(
    xInEmergencyStop := PLC_PRG.DInput1.xDI1,
    xInError := PLC_PRG.DInput1.xDI5,
    xInEnable := Gr.xIN_Run,
    xInRun := Gr.xIN_Run,
    iInPVSpeed := SEL(KM_Gr, 0, 100),
    rInKMapSpeed := 1,
    xInEnRotationSensor := FALSE,
    xInAckError := PLC_PRG.xAck); // Motor
Gr.xOUT_Error := Grohot.xOutError;
Gr.xOUT_Work := Grohot.xOutWork;
Gr.xOUT_Ready := Grohot.xOutReady;
Gr.xOUT_Run := Grohot.xOutRun;
K0.iOUT_PVSpeed := Grohot.iOutPVSpeed;
// КОНВЕЕР ПОДАЧИ
iSP_Podacha := REAL_TO_INT(INT_TO_REAL(PD.iMODBUS_SPSpeed) * 0.2);
Podacha(
    xInEmergencyStop := PLC_PRG.DInput1.xDI1,
    xInError := PLC_PRG.DInput1.xDI4,
    xInEnable := PD.xIN_Run,
    xInRun := PD.xIN_Run,
    iInPVSpeed := PD.iMODBUS_PVSpeed,
    rInKMapSpeed := 0.2,
    iInSPSpeed := iSP_Podacha,
    iInCurrent := PD.iMODBUS_Iengie,
    rInMapCurrent := 0.1,
    xInEnRotationSensor := PD_xIN_EnCtrlSensor,
    xInRotationSensor := PLC_PRG.DInput1.xDI19,
    iInTimeRotationCtrl := PD_iIN_SPRotatTimeMS,
    xInAckError := PLC_PRG.xAck); // Motor
PD.xOUT_Error := Podacha.xOutError;
PD.xOUT_Work := Podacha.xOutWork;
PD.xOUT_Ready := Podacha.xOutReady;
PD.xMODBUS_Run := Podacha.xOutRun;
PD.iOUT_PVSpeed := Podacha.iOutPVSpeed;
PD.rOUT_Current := Podacha.rOutCurrent;
PD.iOUT_PVRotation := Podacha.iOutPVRotationTime;
// Барабан
Baraban(
    xInEmergencyStop := PLC_PRG.DInput1.xDI1,
    xInError := PLC_PRG.DInput1.xDI10,
    xInEnable := BR.xIN_Run,
    xInRun := BR.xIN_Run,
    xInEnRotationSensor := FALSE,
    xInAckError := PLC_PRG.xAck); // Motor
BR.xOUT_Error := Baraban.xOutError;
BR.xOUT_Work := Baraban.xOutWork;
BR.xOUT_Ready := Baraban.xOutReady;
BR.xOUT_Run := Baraban.xOutRun;
BR.rOUT_PVSpeed := INT_TO_REAL(BR.iIN_MODBUS_PVSpeed) * 0.1;
// Элеватор
Elevator(
    xInEmergencyStop := PLC_PRG.DInput1.xDI1,
    xInError := PLC_PRG.DInput1.xDI11,
    xInEnable := EL.xIN_Run,
    xInRun := EL.xIN_Run,
    iInPVSpeed := EL.iIN_MODBUS_PVSpeed,
    rInKMapSpeed := 0.02,
    iInSPSpeed := EL_iIN_SPSpeed,
    iInCurrent := EL.iIN_MODBUS_Iengie,
    rInMapCurrent := 0.01,
    xInEnRotationSensor := EL_xIN_EnCtrlSensor,
    xInRotationSensor := PLC_PRG.DInput1.xDI20,
    iInTimeRotationCtrl := EL_iIN_SPRotatTimeMS,
    xInAckError := PLC_PRG.xAck); // Motor
EL.xOUT_Error := Elevator.xOutError;
EL.xOUT_Work := Elevator.xOutWork;
EL.xOUT_Ready := Elevator.xOutReady;
EL.xOUT_MODBUS_Run := Elevator.xOutRun;
EL.iOUT_PVSpeed := Elevator.iOutPVSpeed;
EL.iOUT_MODBUS_SPSpeed := Elevator.iOutSPSpeedFVVV;
EL.rOUT_Current := Elevator.rOutCurrent;
EL.iOUT_PVRotation := Elevator.iOutPVRotationTime;
// Дымосос
Dedusting(
    xInEmergencyStop := PLC_PRG.DInput1.xDI1,
    xInError := PLC_PRG.DInput1.xDI11,
    xInEnable := Ded.xIN_Run,
    xInRun := Ded.xIN_Run,
    iInPVSpeed := Ded.iIN_MODBUS_PVSpeed,
    rInKMapSpeed := 0.02,
    iInSPSpeed := Ded_iIN_SPSpeed,
    iInCurrent := Ded.iIN_MODBUS_Iengie,
    rInMapCurrent := 0.01,
    xInEnRotationSensor := FALSE,
    xInAckError := PLC_PRG.xAck); // Motor
Ded.xOUT_Error := Dedusting.xOutError;
Ded.xOUT_Work := Dedusting.xOutWork;
Ded.xOUT_Ready := Dedusting.xOutReady;
Ded.xOUT_MODBUS_Run := Dedusting.xOutRun;
Ded.iOUT_PVSpeed := Dedusting.iOutPVSpeed;
Ded.iOUT_MODBUS_SPSpeed := Dedusting.iOutSPSpeedFVVV;
Ded.rOUT_Current := Dedusting.rOutCurrent;
// Вибратор
VIBRATOR(
    ENABLE := xVibEnable,
    TIMELOW := INT_TO_TIME(iVibPause * 1000),
    TIMEHIGH := INT_TO_TIME(iVibWork * 1000)); // BLINK
xVibRun := VIBRATOR.OUT AND xVibEnable AND EL.xOUT_Work OR xVibTEST;
// Вентилятор
xVentWork := NOT (xVentWorkBit1 AND xVentWorkBit2);
rOutVentPVSpeed := INT_TO_REAL(iInMBVentPVSpeed) * 0.02;
// === ГОРЕЛКА ===
AckGor(IN := xGorAckButton, PT := t#2s); // TOF
xGorAck := AckGor.Q;
xGorFaultRS(SET := xGorFault, RESET1 := xGorAck); // RS
xGorRun := (xGorOprob AND NOT xGorRunAUTO AND NOT FALSE OR xGorRunAUTO AND NOT FALSE AND xGorSwitchRun) AND PLC_PRG.DInput1.xDI1;
rOutGorPVTemp := INT_TO_REAL(iInMBGorPVTemp) * 0.1;
rOutGorSPTemp := INT_TO_REAL(iInMBGorSPTemp) * 0.1;
rOutDedPVTemp := INT_TO_REAL(iInMBDedPVTemp) * 0.1;
Drobilka(
    xInEmergencyStop := PLC_PRG.DInput1.xDI1,
    xInError := PLC_PRG.DInput2.xDI6,
    xInEnable := xDrobRun,
    xInRun := xDrobRun,
    xInEnRotationSensor := FALSE,
    xInAckError := PLC_PRG.xAck); // Motor
xDrob_OUT_Error := Drobilka.xOutError;
xDrob_OUT_Work := Drobilka.xOutWork;
xDrob_OUT_Ready := Drobilka.xOutReady;
xDrob_OUT_Run := Drobilka.xOutRun;

END_PROGRAM

// Device/Application/Motor
FUNCTION_BLOCK Motor
VAR_INPUT
	//Аварийный стоп
	xInEmergencyStop: BOOL;
	// Ошибка преобразователя
	xInError: BOOL;
	// Режим Использования
	xInEnable: BOOL;
	// Пуск
	xInRun: BOOL;
	
	//факт обороты
	iInPVSpeed: INT;
	//Коэф.маштабирования оборотов
	rInKMapSpeed: REAL;
	//Задание оборотов (0-100%)
	iInSPSpeed: INT;
	
	// Ток двигателя
	iInCurrent: INT;
	// Коэф маштабирования тока
	rInMapCurrent: REAL;
	
	// Контроль вращения Включить
	xInEnRotationSensor: BOOL;
	// Датчик контроля вращения
	xInRotationSensor: BOOL;
	// Время контороля вращения
	iInTimeRotationCtrl: INT;
	
	// Вход Подтвердить ошибку
	xInAckError: BOOL;
END_VAR
VAR_OUTPUT
	// Ошибка
	xOutError: BOOL;
	// Двигатель работает
	xOutWork: BOOL;
	//Готовность
	xOutReady: BOOL;
	// Команда ПУСК
	xOutRun: BOOL;
	

	//Факт частота вращения(0-100%)
	iOutPVSpeed: INT;
	// Задание частоты вращения(0-10000) для ПЧ
	iOutSPSpeedFVVV:INT;
	
	// Ток двигателя
	rOutCurrent: REAL;
	
	//Факт время оборота, мс
	iOutPVRotationTime: INT;
END_VAR

VAR
	// Готовность
	xReady: BOOL;
	// Команда Пуск
	xRun: BOOL;
	// Работает
	xWork1: BOOL;
	// Фактическое время вращения
	PVRotationTimeMilliSecund: TIME;
	// Заданное время вращения
	SPRotationTimeMilliSecund: TIME;

	xPFront: BOOL;
	xNFront: BOOL;
	T2: TON;
	T1: TON;
	xC: BOOL;
	rTemp1: REAL;
	rTemp2: REAL;
	xTemp1: BOOL;
	xFirstRun: BOOL;
	T0: TON;
	SPRotationTimeMilliSecund3: TIME;
	PVRotationTimeMilliSecund3: TIME;
	xStartNoRotation: BOOL;
	xNoRation: BOOL;
	xExtError: BOOL;
END_VAR
VAR // added by the converter: edge detectors and wires of the graphical bodies
    _rt1, _rt2, _rt3 : R_TRIG;
    _ft1, _ft2, _ft3 : F_TRIG;
    _w1, _w2 : BOOL;
END_VAR

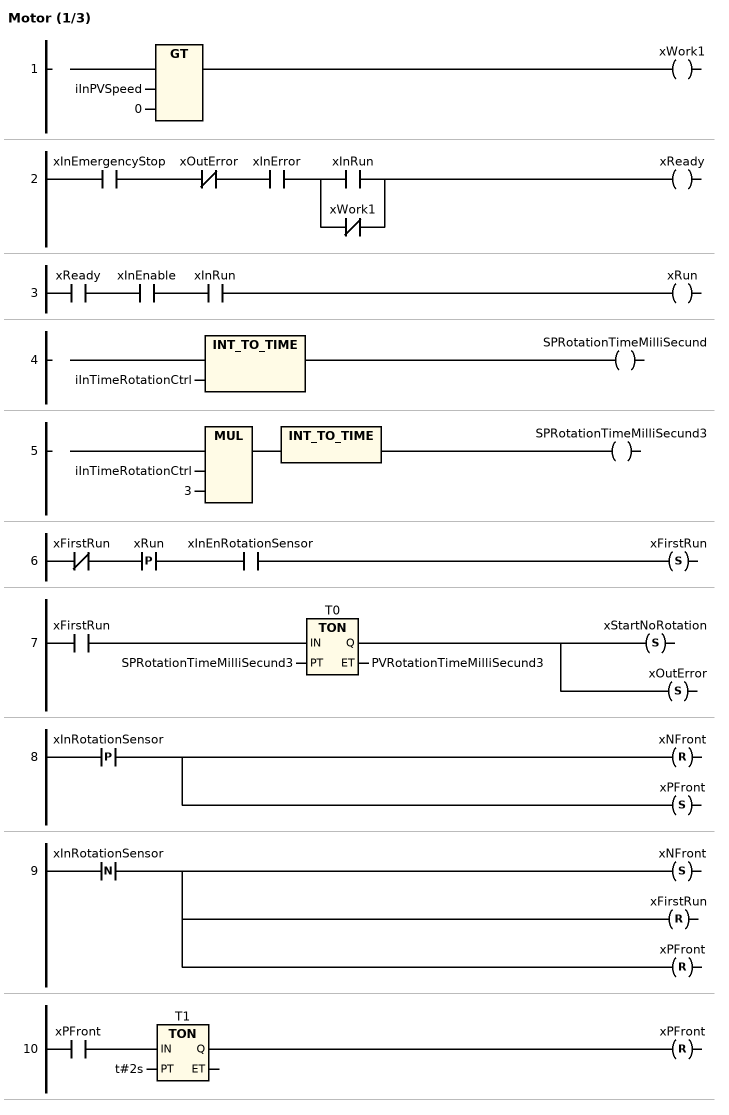
// NETWORK 1
xWork1 := iInPVSpeed > 0;

// NETWORK 2
xReady := xInEmergencyStop AND NOT xOutError AND xInError AND (xInRun OR NOT xWork1);

// NETWORK 3
xRun := xReady AND xInEnable AND xInRun;

// NETWORK 4
SPRotationTimeMilliSecund := INT_TO_TIME(iInTimeRotationCtrl);

// NETWORK 5
SPRotationTimeMilliSecund3 := INT_TO_TIME(iInTimeRotationCtrl * 3);

// NETWORK 6
_rt1(CLK := xRun);
xFirstRun S= NOT xFirstRun AND _rt1.Q AND xInEnRotationSensor;

// NETWORK 7
T0(IN := xFirstRun, PT := SPRotationTimeMilliSecund3, ET => PVRotationTimeMilliSecund3); // TON
xStartNoRotation S= T0.Q;
xOutError S= T0.Q;

// NETWORK 8
_rt2(CLK := xInRotationSensor);
xNFront R= _rt2.Q;
xPFront S= _rt2.Q;

// NETWORK 9
_ft1(CLK := xInRotationSensor);
xNFront S= _ft1.Q;
xFirstRun R= _ft1.Q;
xPFront R= _ft1.Q;

// NETWORK 10
T1(IN := xPFront, PT := t#2s); // TON
xPFront R= T1.Q;

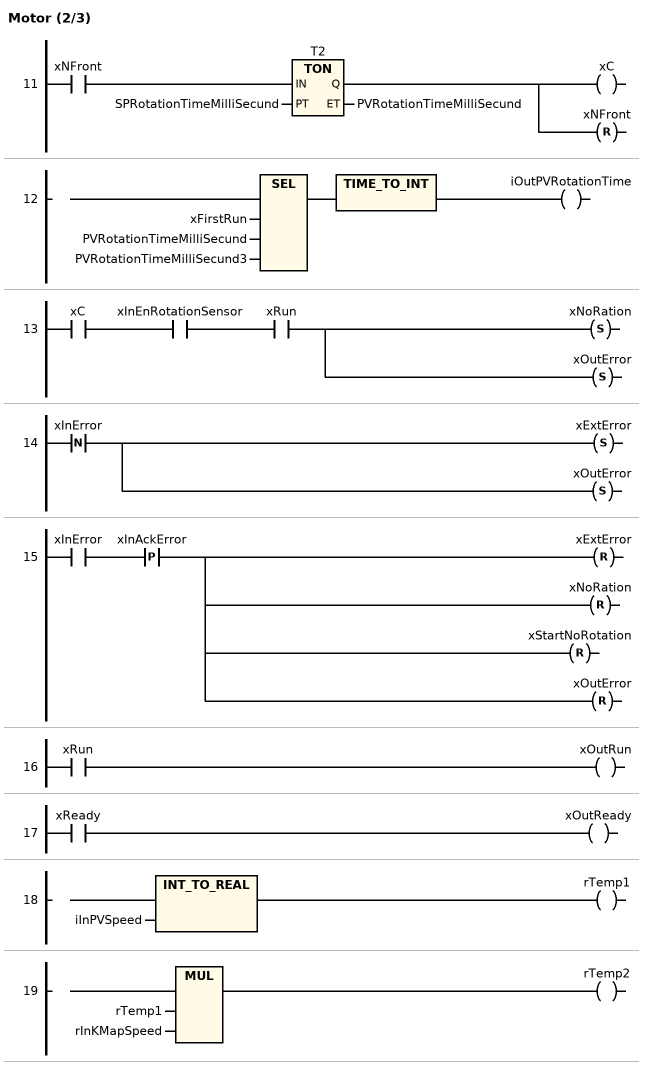
// NETWORK 11
T2(IN := xNFront, PT := SPRotationTimeMilliSecund, ET => PVRotationTimeMilliSecund); // TON
xC := T2.Q;
xNFront R= T2.Q;

// NETWORK 12
iOutPVRotationTime := TIME_TO_INT(SEL(xFirstRun, PVRotationTimeMilliSecund, PVRotationTimeMilliSecund3));

// NETWORK 13
_w1 := xC AND xInEnRotationSensor AND xRun;
xNoRation S= _w1;
xOutError S= _w1;

// NETWORK 14
_ft2(CLK := xInError);
xExtError S= _ft2.Q;
xOutError S= _ft2.Q;

// NETWORK 15
_rt3(CLK := xInAckError);
_w2 := xInError AND _rt3.Q;
xExtError R= _w2;
xNoRation R= _w2;
xStartNoRotation R= _w2;
xOutError R= _w2;

// NETWORK 16
xOutRun := xRun;

// NETWORK 17
xOutReady := xReady;

// NETWORK 18
rTemp1 := INT_TO_REAL(iInPVSpeed);

// NETWORK 19
rTemp2 := rTemp1 * rInKMapSpeed;

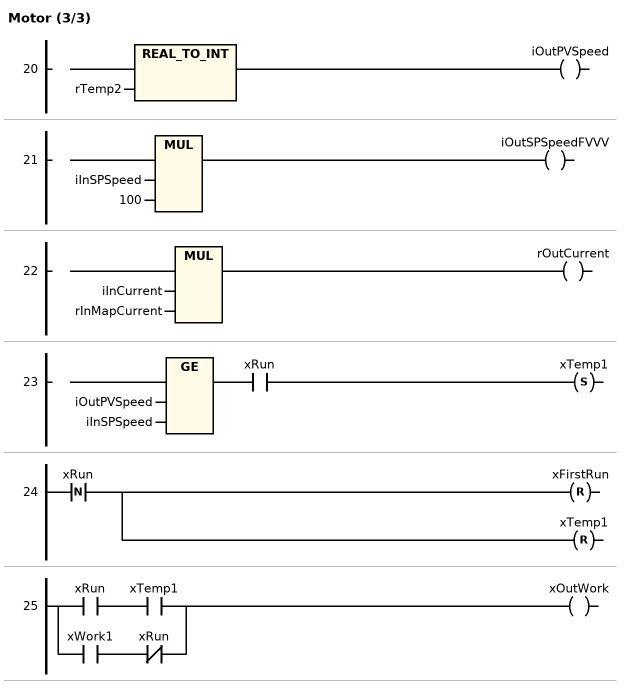
// NETWORK 20
iOutPVSpeed := REAL_TO_INT(rTemp2);

// NETWORK 21
iOutSPSpeedFVVV := iInSPSpeed * 100;

// NETWORK 22
rOutCurrent := iInCurrent * rInMapCurrent;

// NETWORK 23
xTemp1 S= iOutPVSpeed >= iInSPSpeed AND xRun;

// NETWORK 24
_ft3(CLK := xRun);
xFirstRun R= _ft3.Q;
xTemp1 R= _ft3.Q;

// NETWORK 25
xOutWork := xRun AND xTemp1 OR xWork1 AND NOT xRun;

END_FUNCTION_BLOCK

// Device/Application/CountWebCli
PROGRAM CountWebCli
VAR
	pClient: POINTER TO VisuElems.VisuStructClientData;
	iCountActivWebVisus: INT;
	xAlarm: BOOL;
END_VAR

iCountActivWebVisus:=0;
xAlarm:=FALSE;

VisuElems.VisuElemBase.g_ClientManager.BeginIteration();

WHILE (pClient:=VisuElems.VisuElemBase.g_ClientManager.GetNextClient())<>0 DO
	IF pClient^.GlobalData.ClientType = VisuElems.Visu_ClientType.Webvisualization THEN
		iCountActivWebVisus:=iCountActivWebVisus+1;
		xAlarm:=TRUE;
	END_IF
END_WHILE

END_PROGRAM

// Device/Application/Chain
PROGRAM Chain
VAR
	ReadyRun: BOOL:=FALSE;
	Run: BOOL:=FALSE;
	EmerSTOP: BOOL;
	Stop5: BOOL;	

	Step: INT:=0;

	TMR990: TON;
	Stoped995: BOOL;
	Runed5: BOOL;
	Stop10: BOOL;
	Runed10: BOOL;
	Stop: BOOL;
	Stoped990: BOOL;
	TMR5: TON;
	Stop15: BOOL;
	Runed15: BOOL;
	Stoped985: BOOL;
	Stop20: BOOL;
	Runed20: BOOL;
	TMR980: TON;
	Stop25: BOOL;
	Runed25: BOOL;
	TMR975: TON;
	Stop30: BOOL;
	TMRWork: TON;
	TMR970: TON;
	xLampPUSK: BOOL;
END_VAR

//IF <condition> THEN
//    <statements>
//( ELSIF <condition> THEN
//        <statements> )*
//( ELSE
//        <statements> )?
//END_IF;
// ( ... )* None, once or several times
// ( ... )? Optional

//	TMR995 (IN:=Step=995 AND NOT(TMR995.Q), PT:=T#5S);
//	IF TMR995.Q THEN
//		Step:=0;
//	END_IF

EmerSTOP:= NOT(PLC_PRG.DInput1.xDI1);

ReadyRun:= PLC_PRG.DInput1.xDI1 // ававрийный стоп
			AND MECH.K40.xOUT_Ready
			AND MECH.K25.xOUT_Ready
			AND MECH.K10.xOUT_Ready
			AND MECH.K0.xOUT_Ready
			AND MECH.Gr.xOUT_Ready
			AND MECH.PD.xOUT_Ready
			AND MECH.Ded.xOUT_Ready
			AND MECH.BR.xOUT_Ready
			AND MECH.EL.xOUT_Ready
			AND PLC_PRG.DInput2.xDI2 //шибер закрыт
			AND NOT(MECH.xGorOprob)
			AND MECH.xDrob_OUT_Ready;
			
Stop:=NOT(PLC_PRG.DInput1.xDI14);

			
Run:= PLC_PRG.DInput1.xDI13 
		AND PLC_PRG.DInput1.xDI14;

Runed5:= MECH.K40.xOUT_Work
		AND MECH.K25.xOUT_Work
		AND MECH.K10.xOUT_Work
		AND MECH.K0.xOUT_Work
		AND MECH.Ded.xOUT_Work
		AND MECH.xDrob_OUT_Work;

Runed10:= MECH.Gr.xOUT_Work;

Runed15:= MECH.PD.xOUT_Work;

Runed20:= MECH.BR.xOUT_Work;

Runed25:= MECH.EL.xOUT_Work;		

Stop5:=   MECH.K40.xOUT_Error
		OR MECH.K25.xOUT_Error
		OR MECH.K10.xOUT_Error
		OR MECH.K0.xOUT_Error
		OR MECH.Ded.xOUT_Error
		OR MECH.xDrob_OUT_Error;
		
Stop10:= MECH.Gr.xOUT_Error;

Stop15:= MECH.PD.xOUT_Error;

Stop20:= MECH.BR.xOUT_Error;

Stop25:= MECH.EL.xOUT_Error;

Stoped985:=//NOT(MECH.K40.xOUT_Work)
		//AND NOT(MECH.K25.xOUT_Work)
		//AND NOT(MECH.K10.xOUT_Work)
		//AND NOT(MECH.K0.xOUT_Work)
		//AND NOT(MECH.Ded.xOUT_Work)
		//AND NOT(MECH.Gr.xOUT_Work)
			NOT(MECH.PD.xOUT_Work)
		AND NOT(MECH.BR.xOUT_Work)
		AND NOT(MECH.EL.xOUT_Work);
		//AND NOT(MECH.Gorelka.xOUT_Work);
		
Stoped995:=NOT(MECH.K40.xOUT_Work)
		AND NOT(MECH.K25.xOUT_Work)
		AND NOT(MECH.K10.xOUT_Work)
		AND NOT(MECH.K0.xOUT_Work)
		AND NOT(MECH.Ded.xOUT_Work)
		AND NOT(MECH.Gr.xOUT_Work)
		AND NOT(MECH.PD.xOUT_Work)
		AND NOT(MECH.BR.xOUT_Work)
		AND NOT(MECH.EL.xOUT_Work)
		AND NOT(MECH.xDrob_OUT_Work);
		//AND NOT(MECH.Gorelka.xOUT_Work);
		


///===============================================================================================================================

IF Step=0 THEN
	IF ReadyRun THEN
		IF Run THEN
			Step:=5;
		END_IF;
		ELSE 
		Step:=1;
	END_IF;
ELSIF Step=1 THEN
	IF ReadyRun THEN
		Step:=0;
	END_IF

// ЗАПУСК КОНВЕЕРОВ ФРАКЦИЙ и Д/С, ДРОБИЛКИ	
ELSIF Step=5 THEN
	MECH.K40.xIN_Run:=TRUE;
	MECH.K25.xIN_Run:=TRUE;
	MECH.K10.xIN_Run:=TRUE;
	MECH.K0.xIN_Run:=TRUE;
	MECH.Ded.xIN_Run:=TRUE;
	MECH.xDrobRun:=TRUE;
	xLampPUSK:=TRUE;
	IF Stop5 OR Stop THEN
		Step:=995;	
	END_IF;
	IF EmerSTOP THEN
		Step:=1000;
	END_IF;
	IF Runed5 THEN
		Step:=10;		
	END_IF;

// ЗАПУСК ГРОХОТА	
ELSIF Step=10 THEN	
	MECH.Gr.xIN_Run:=TRUE;

	IF Stop5 THEN
		Step:=995;	
	END_IF;
	
	IF Stop10 OR Stop THEN
		Step:=990;	
	END_IF;
	IF EmerSTOP THEN
		Step:=1000;
	END_IF;
	
	TMR5 (IN:=Step=10 AND NOT(TMR5.Q), PT:=T#10S);
	IF Runed10 AND TMR5.Q THEN
		Step:=15;		
	END_IF;


// ЗАПУСК ПОДАЧИ 	
ELSIF Step=15 THEN	
	MECH.PD.xIN_Run:=TRUE;

	IF Stop5 THEN
		Step:=995;	
	END_IF;
	
	IF Stop10 THEN
		Step:=990;	
	END_IF;
	
	IF Stop15 OR Stop THEN
		Step:=985;	
	END_IF;
	
	IF EmerSTOP THEN
		Step:=1000;
	END_IF;
	
	IF Runed15 THEN
		Step:=20;		
	END_IF;
	
	
	
// ЗАПУСК БАРАБАНА И ГОРЕЛКИ
ELSIF Step=20 THEN	
	MECH.BR.xIN_Run:=TRUE;
	MECH.xGorRunAUTO:=TRUE;

	IF Stop5 THEN
		Step:=995;	
	END_IF;
	
	IF Stop10 THEN
		Step:=990;	
	END_IF;
	
	IF Stop15 THEN
		Step:=985;	
	END_IF;
	
	IF Stop20 OR Stop THEN
		Step:=980;	
	END_IF;
	
	IF EmerSTOP THEN
		Step:=1000;
	END_IF;
	
	IF Runed20 THEN
		Step:=25;		
	END_IF;
	
// ЗАПУСК ЭЛЕВАТОРА
ELSIF Step=25 THEN	
	MECH.EL.xIN_Run:=TRUE;
	
	IF Stop5 THEN
		Step:=995;	
	END_IF;
	
	IF Stop10 THEN
		Step:=990;	
	END_IF;
	
	IF Stop15 THEN
		Step:=985;	
	END_IF;
	
	IF Stop20 THEN
		Step:=980;	
	END_IF;
	
	IF Stop25 OR Stop THEN
		Step:=975;	
	END_IF
	
	IF EmerSTOP THEN
		Step:=1000;
	END_IF;
	
	IF Runed25 THEN
		Step:=30;		
	END_IF;
	
// ЗАПУСК ВИБРАТОРА и ТАЙМЕРА РАБОТЫ
ELSIF Step=30 THEN	
	MECH.xVibRunAUTO:=TRUE;
		
	IF Stop5 THEN
		Step:=995;	
	END_IF;
	
	IF Stop10 THEN
		Step:=990;	
	END_IF;
	
	IF Stop15 THEN
		Step:=985;	
	END_IF;
	
	IF Stop20 THEN
		Step:=980;	
	END_IF;
	
	IF Stop25 THEN
		Step:=975;	
	END_IF
	
	IF Stop THEN
		Step:=970;	
	END_IF
	
	IF EmerSTOP THEN
		Step:=1000;
	END_IF;
	
	TMRWork (IN:=Step=30, PT:=T#1D);
		
//////////////=========================================

// ОСТАНОВКА ВИБРАТОРА
ELSIF Step=970 THEN
	//MECH.K40.xIN_Run:=FALSE;
	//MECH.K25.xIN_Run:=FALSE;
	//MECH.K10.xIN_Run:=FALSE;
	//MECH.K0.xIN_Run:=FALSE;
	//MECH.Ded.xIN_Run:=FALSE;
	//MECH.Gr.xIN_Run:=FALSE;
	//MECH.PD.xIN_Run:=FALSE;
	//MECH.BR.xIN_Run:=FALSE;
	//MECH.EL.xIN_Run:=FALSE;
	//MECH.Gorelka.xIN_Run:=FALSE;
	MECH.xVibRunAUTO:=FALSE;
	xLampPUSK:=FALSE;
	
	TMR970 (IN:=Step=970 AND NOT(TMR970.Q), PT:=T#10S);
	IF TMR970.Q THEN
		Step:=975;
	END_IF

// ОСТАНОВКА ЭЛЕВАТОРА
ELSIF Step=975 THEN
	//MECH.K40.xIN_Run:=FALSE;
	//MECH.K25.xIN_Run:=FALSE;
	//MECH.K10.xIN_Run:=FALSE;
	//MECH.K0.xIN_Run:=FALSE;
	//MECH.Ded.xIN_Run:=FALSE;
	//MECH.Gr.xIN_Run:=FALSE;
	//MECH.PD.xIN_Run:=FALSE;
	//MECH.BR.xIN_Run:=FALSE;
	MECH.EL.xIN_Run:=FALSE;
	//MECH.xGorRunAUTO:=FALSE;
	MECH.xVibRunAUTO:=FALSE;
	xLampPUSK:=FALSE;
	
	TMR975 (IN:=Step=975 AND NOT(TMR975.Q), PT:=T#10S);
	IF TMR975.Q THEN
		Step:=980;
	END_IF
	
	
// ОСТАНОВКА БАРАБАНА
ELSIF Step=980 THEN
	//MECH.K40.xIN_Run:=FALSE;
	//MECH.K25.xIN_Run:=FALSE;
	//MECH.K10.xIN_Run:=FALSE;
	//MECH.K0.xIN_Run:=FALSE;
	//MECH.Ded.xIN_Run:=FALSE;
	//MECH.Gr.xIN_Run:=FALSE;
	//MECH.PD.xIN_Run:=FALSE;
	MECH.BR.xIN_Run:=FALSE;
	MECH.EL.xIN_Run:=FALSE;
	MECH.xGorRunAUTO:=FALSE;
	MECH.xVibRunAUTO:=FALSE;
	xLampPUSK:=FALSE;
	
	TMR980 (IN:=Step=980 AND NOT(TMR980.Q), PT:=T#10S);
	IF TMR980.Q THEN
		Step:=985;
	END_IF
	//IF Stoped985 THEN
	//	Step:=985;
	//END_IF
	
// ОСТАНОВКА ПОДАЧИ
ELSIF Step=985 THEN
	//MECH.K40.xIN_Run:=FALSE;
	//MECH.K25.xIN_Run:=FALSE;
	//MECH.K10.xIN_Run:=FALSE;
	//MECH.K0.xIN_Run:=FALSE;
	//MECH.Ded.xIN_Run:=FALSE;
	//MECH.Gr.xIN_Run:=FALSE;
	MECH.PD.xIN_Run:=FALSE;
	MECH.BR.xIN_Run:=FALSE;
	MECH.EL.xIN_Run:=FALSE;
	MECH.xGorRunAUTO:=FALSE;
	MECH.xVibRunAUTO:=FALSE;
	xLampPUSK:=FALSE;
	
	IF Stoped985 THEN
		Step:=990;
	END_IF

// ОСТАНОВКА ГРОХОТА
ELSIF Step=990 THEN
	//MECH.K40.xIN_Run:=FALSE;
	//MECH.K25.xIN_Run:=FALSE;
	//MECH.K10.xIN_Run:=FALSE;
	//MECH.K0.xIN_Run:=FALSE;
	//MECH.Ded.xIN_Run:=FALSE;
	MECH.Gr.xIN_Run:=FALSE;
	MECH.PD.xIN_Run:=FALSE;
	MECH.BR.xIN_Run:=FALSE;
	MECH.EL.xIN_Run:=FALSE;
	MECH.xGorRunAUTO:=FALSE;
	MECH.xVibRunAUTO:=FALSE;
	xLampPUSK:=FALSE;
	
	TMR990 (IN:=Step=990 AND NOT(TMR990.Q), PT:=T#30S);
	IF TMR990.Q THEN
		Step:=995;
	END_IF

// ОСТАНОВКА КОНВЕЕРОВ И Д/С	
ELSIF Step=995 THEN
	MECH.K40.xIN_Run:=FALSE;
	MECH.K25.xIN_Run:=FALSE;
	MECH.K10.xIN_Run:=FALSE;
	MECH.K0.xIN_Run:=FALSE;
	MECH.Ded.xIN_Run:=FALSE;
	MECH.Gr.xIN_Run:=FALSE;
	MECH.PD.xIN_Run:=FALSE;
	MECH.BR.xIN_Run:=FALSE;
	MECH.EL.xIN_Run:=FALSE;
	MECH.xGorRunAUTO:=FALSE;
	MECH.xVibRunAUTO:=FALSE;
	MECH.xDrobRun:=FALSE;
	xLampPUSK:=FALSE;
	IF Stoped995 THEN
		Step:=0;
	END_IF

// АВАРИЙНЫЙ СТОП!!	
ELSIF Step=1000 THEN
	MECH.K40.xIN_Run:=FALSE;
	MECH.K25.xIN_Run:=FALSE;
	MECH.K10.xIN_Run:=FALSE;
	MECH.K0.xIN_Run:=FALSE;
	MECH.Ded.xIN_Run:=FALSE;
	MECH.Gr.xIN_Run:=FALSE;
	MECH.PD.xIN_Run:=FALSE;
	MECH.BR.xIN_Run:=FALSE;
	MECH.EL.xIN_Run:=FALSE;
	MECH.xGorRunAUTO:=FALSE;
	MECH.xVibRunAUTO:=FALSE;
	MECH.xDrobRun:=FALSE;
	xLampPUSK:=FALSE;
	IF	PLC_PRG.xAck AND Stoped995 THEN
		Step:=0;
	END_IF		
END_IF

END_PROGRAM

// Device/Application/VFrADiag
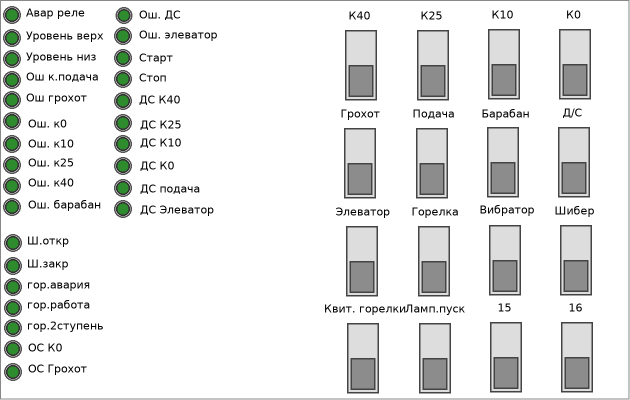
VISUALIZATION VFrADiag  // 630x400, background image ImagePool.fonFreame
    Lamp1 (2,5 20x20), variable: PLC_PRG.DInput1.xDI1, style: Lamp-Lamp1-Green
    Lamp1 (2,28 20x20), variable: PLC_PRG.DInput1.xDI2, style: Lamp-Lamp1-Green
    Lamp1 (2,49 20x20), variable: PLC_PRG.DInput1.xDI3, style: Lamp-Lamp1-Green
    Lamp1 (2,70 20x20), variable: PLC_PRG.DInput1.xDI4, style: Lamp-Lamp1-Green
    Lamp1 (2,90 20x20), variable: PLC_PRG.DInput1.xDI5, style: Lamp-Lamp1-Green
    Lamp1 (2,111 20x20), variable: PLC_PRG.DInput1.xDI6, style: Lamp-Lamp1-Green
    Lamp1 (2,134 20x20), variable: PLC_PRG.DInput1.xDI7, style: Lamp-Lamp1-Green
    Lamp1 (2,155 20x20), variable: PLC_PRG.DInput1.xDI8, style: Lamp-Lamp1-Green
    Lamp1 (2,176 20x20), variable: PLC_PRG.DInput1.xDI9, style: Lamp-Lamp1-Green
    Lamp1 (2,197 20x20), variable: PLC_PRG.DInput1.xDI10, style: Lamp-Lamp1-Green
    Lamp1 (113,6 22x19), variable: PLC_PRG.DInput1.xDI11, style: Lamp-Lamp1-Green
    Lamp1 (113,26 20x20), variable: PLC_PRG.DInput1.xDI12, style: Lamp-Lamp1-Green
    Lamp1 (113,48 20x20), variable: PLC_PRG.DInput1.xDI13, style: Lamp-Lamp1-Green
    Lamp1 (113,69 20x20), variable: PLC_PRG.DInput1.xDI14, style: Lamp-Lamp1-Green
    Lamp1 (113,91 20x20), variable: PLC_PRG.DInput1.xDI15, style: Lamp-Lamp1-Green
    Lamp1 (113,113 20x20), variable: PLC_PRG.DInput1.xDI16, style: Lamp-Lamp1-Green
    Lamp1 (113,134 20x20), variable: PLC_PRG.DInput1.xDI17, style: Lamp-Lamp1-Green
    Lamp1 (113,156 20x20), variable: PLC_PRG.DInput1.xDI18, style: Lamp-Lamp1-Green
    Lamp1 (113,178 20x20), variable: PLC_PRG.DInput1.xDI19, style: Lamp-Lamp1-Green
    Lamp1 (113,199 20x20), variable: PLC_PRG.DInput1.xDI20, style: Lamp-Lamp1-Green
    Label (23,-2 66x30), "Авар реле"
    Label (23,62 86x30), "Ош к.подача"
    Label (23,83 83x30), "Ош грохот"
    Label (25,148 61x30), "Ош. к25"
    Label (25,168 62x30), "Ош. к40"
    Label (25,109 63x30), "Ош. к0"
    Label (136,20 79x30), "Ош. элеватор"
    Label (136,43 40x30), "Старт"
    Label (136,63 40x30), "Стоп"
    Label (136,85 66x30), "ДС К40"
    Label (25,190 123x30), "Ош. барабан"
    Label (136,0 53x30), "Ош. ДС"
    Label (23,21 93x30), "Уровень верх"
    Label (23,42 89x30), "Уровень низ"
    Label (25,129 63x30), "Ош. к10"
    Label (137,110 57x30), "ДС К25"
    Label (137,128 57x30), "ДС К10"
    Label (137,151 40x30), "ДС К0"
    Label (137,174 64x30), "ДС подача"
    Label (137,195 77x30), "ДС Элеватор"
    DipSwitch (328,323 70x70), variable: PLC_PRG.DOutput1.xDO13, input disabled if: TRUE, behaviour: TOGGLE, style: Switch-DipSwitch-Gray
    Label (318,299 94x20), "Квит. горелки"
    DipSwitch (400,323 70x70), variable: PLC_PRG.DOutput1.xDO14, input disabled if: TRUE, behaviour: TOGGLE, style: Switch-DipSwitch-Gray
    Label (399,299 72x20), "Ламп.пуск"
    DipSwitch (471,322 70x70), variable: PLC_PRG.DOutput1.xDO15, input disabled if: TRUE, behaviour: TOGGLE, style: Switch-DipSwitch-Gray
    Label (488,298 33x20), "15"
    DipSwitch (542,322 70x70), variable: PLC_PRG.DOutput1.xDO16, input disabled if: TRUE, behaviour: TOGGLE, style: Switch-DipSwitch-Gray
    Label (559,298 33x20), "16"
    DipSwitch (326,30 70x70), variable: MECH.K40.xIN_Run, input disabled if: TRUE, behaviour: TOGGLE, style: Switch-DipSwitch-Gray
    Label (343,6 33x20), "К40"
    DipSwitch (398,30 70x70), variable: MECH.K25.xIN_Run, input disabled if: TRUE, behaviour: TOGGLE, style: Switch-DipSwitch-Gray
    Label (415,6 33x20), "К25"
    DipSwitch (469,29 70x70), variable: MECH.K10.xIN_Run, input disabled if: TRUE, behaviour: TOGGLE, style: Switch-DipSwitch-Gray
    Label (486,5 33x20), "К10"
    DipSwitch (540,29 70x70), variable: MECH.K0.xIN_Run, input disabled if: TRUE, behaviour: TOGGLE, style: Switch-DipSwitch-Gray
    Label (557,5 33x20), "К0"
    DipSwitch (325,128 70x70), variable: MECH.Gr.xIN_Run, input disabled if: TRUE, behaviour: TOGGLE, style: Switch-DipSwitch-Gray
    Label (338,104 45x20), "Грохот"
    DipSwitch (397,128 70x70), variable: MECH.PD.xIN_Run, input disabled if: TRUE, behaviour: TOGGLE, style: Switch-DipSwitch-Gray
    Label (407,104 53x20), "Подача"
    DipSwitch (468,127 70x70), variable: MECH.BR.xIN_Run, input disabled if: TRUE, behaviour: TOGGLE, style: Switch-DipSwitch-Gray
    Label (477,104 57x20), "Барабан"
    DipSwitch (539,127 70x70), variable: MECH.Ded.xIN_Run, input disabled if: TRUE, behaviour: TOGGLE, style: Switch-DipSwitch-Gray
    Label (556,103 33x20), "Д/С"
    DipSwitch (327,226 70x70), variable: MECH.EL.xIN_Run, input disabled if: TRUE, behaviour: TOGGLE, style: Switch-DipSwitch-Gray
    Label (328,202 70x20), "Элеватор"
    DipSwitch (399,226 70x70), variable: PLC_PRG.DOutput1.xDO10, input disabled if: TRUE, behaviour: TOGGLE, style: Switch-DipSwitch-Gray
    Label (405,202 60x20), "Горелка"
    DipSwitch (470,225 70x70), variable: MECH.xVibRun, input disabled if: TRUE, behaviour: TOGGLE, style: Switch-DipSwitch-Gray
    Label (474,200 66x20), "Вибратор"
    DipSwitch (541,225 70x70), variable: PLC_PRG.DOutput1.xDO12, input disabled if: TRUE, behaviour: TOGGLE, style: Switch-DipSwitch-Gray
    Label (543,201 63x20), "Шибер"
    Lamp1 (3,233 20x20), variable: PLC_PRG.DInput2.xDI1, style: Lamp-Lamp1-Green
    Lamp1 (3,256 20x20), variable: PLC_PRG.DInput2.xDI2, style: Lamp-Lamp1-Green
    Lamp1 (3,277 20x20), variable: PLC_PRG.DInput2.xDI3, style: Lamp-Lamp1-Green
    Lamp1 (3,298 20x20), variable: PLC_PRG.DInput2.xDI4, style: Lamp-Lamp1-Green
    Lamp1 (3,318 20x20), variable: PLC_PRG.DInput2.xDI5, style: Lamp-Lamp1-Green
    Lamp1 (3,339 20x20), variable: PLC_PRG.DInput2.xDI6, style: Lamp-Lamp1-Green
    Lamp1 (3,362 20x20), variable: PLC_PRG.DInput2.xDI7, style: Lamp-Lamp1-Green
    Label (24,226 66x30), "Ш.откр"
    Label (24,290 86x30), "гор.работа"
    Label (24,311 83x30), "гор.2ступень"
    Label (24,249 93x30), "Ш.закр"
    Label (24,270 89x30), "гор.авария"
    Label (25,354 83x30), "ОС Грохот"
    Label (25,333 86x30), "ОС К0"
END_VISUALIZATION

// Device/Application/VFr4Baraban
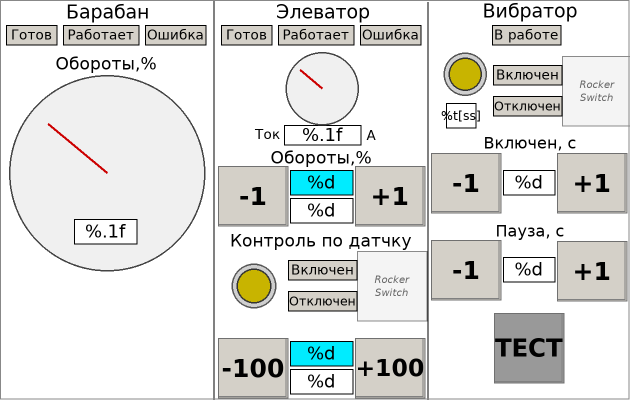
VISUALIZATION VFr4Baraban  // 630x400, background image ImagePool.fonFreame
    Rectangle (503,170 52x25), "%d", text variable: MECH.iVibWork
    Label (455,128 150x30), "Включен, с"
    Button (557,153 70x60), "+1"
        OnMouseClick: execute {
            IF MECH.iVibWork <5 THEN
            	MECH.iVibWork := MECH.iVibWork + 1;
            END_IF;
        }
    Button (431,153 70x60), "-1"
        OnMouseClick: execute {
            IF MECH.iVibWork >1 THEN
            	MECH.iVibWork := MECH.iVibWork - 1;
            END_IF;
        }
    Button (557,241 70x60), "+1"
        OnMouseClick: execute {
            IF MECH.iVibPause <31 THEN
            	MECH.iVibPause := MECH.iVibPause + 1;
            END_IF;
        }
    Rectangle (503,257 52x25), "%d", text variable: MECH.iVibPause
    Label (455,216 150x30), "Пауза, с"
    Button (431,240 70x60), "-1"
        OnMouseClick: execute {
            IF MECH.iVibPause >5 THEN
            	MECH.iVibPause := MECH.iVibPause - 1;
            END_IF;
        }
    Lamp1 (438,49 54x50), variable: MECH.xVibRun, style: Lamp-Lamp1-Yellow
    Label (43,2 130x20), "Барабан"
    Label (24,125 57x19)
    Label (59,56 94x15), "Обороты,%"
    Rectangle (63,25 76x20), "Работает", colour toggle: MECH.BR.xOUT_Work
    Rectangle (145,25 61x20), "Ошибка", colour toggle: MECH.BR.xOUT_Error
    Rectangle (6,25 51x20), "Готов", colour toggle: MECH.BR.xOUT_Ready
    Rectangle (290,198 63x25), "%d", text variable: MECH.EL.iOUT_PVSpeed
    Rectangle (290,170 63x25), "%d", text variable: MECH.EL_iIN_SPSpeed
    Button (355,166 70x60), "+1"
        OnMouseClick: execute {
            IF MECH.EL_iIN_SPSpeed <100 THEN
            	MECH.EL_iIN_SPSpeed := MECH.EL_iIN_SPSpeed + 1;
            END_IF;
        }
    Button (218,166 70x60), "-1"
        OnMouseClick: execute {
            IF MECH.EL_iIN_SPSpeed >5 THEN
            	MECH.EL_iIN_SPSpeed := MECH.EL_iIN_SPSpeed - 1;
            END_IF;
        }
    Label (258,2 130x20), "Элеватор"
    Rectangle (284,125 77x20), "%.1f", text variable: MECH.EL.rOUT_Current
    Label (239,125 57x19), "Ток"
    Label (274,150 94x15), "Обороты,%"
    Rectangle (290,369 63x25), "%d", text variable: MECH.EL.iOUT_PVRotation, colour toggle: MECH.Elevator.xFirstRun
    Rectangle (290,341 63x25), "%d", text variable: MECH.EL_iIN_SPRotatTimeMS
    Button (355,338 70x60), "+100"
        OnMouseClick: execute {
            IF MECH.EL_iIN_SPRotatTimeMS <10000 THEN
            	MECH.EL_iIN_SPRotatTimeMS := MECH.EL_iIN_SPRotatTimeMS + 100;
            END_IF;
        }
    Button (218,338 70x60), "-100"
        OnMouseClick: execute {
            IF MECH.EL_iIN_SPRotatTimeMS >500 THEN
            	MECH.EL_iIN_SPRotatTimeMS := MECH.EL_iIN_SPRotatTimeMS - 100;
            END_IF;
        }
    RockerSwitch (357,251 70x70), variable: MECH.EL_xIN_EnCtrlSensor, behaviour: TOGGLE, style: Switch-RockerSwitch-Yellow
    Meter180 (250,52 144x73), value: MECH.EL.rOUT_Current, style: Meter-Meter180-Green, scale format: %d, scale 0..10
    Rectangle (278,25 76x20), "Работает", colour toggle: MECH.EL.xOUT_Work
    Rectangle (360,25 61x20), "Ошибка", colour toggle: MECH.EL.xOUT_Error
    Rectangle (221,25 51x20), "Готов", colour toggle: MECH.EL.xOUT_Ready
    Label (356,126 30x19), "А"
    Lamp1 (227,260 54x52), variable: PLC_PRG.DInput1.xDI20, style: Lamp-Lamp1-Yellow
    Rectangle (288,260 69x20), "Включен", colour toggle: MECH.EL_xIN_EnCtrlSensor
    Rectangle (288,291 69x20), "Отключен", colour toggle: NOT(MECH.EL_xIN_EnCtrlSensor)
    Label (219,231 204x19), "Контроль по датчку"
    Line (214,401) (214,1)
    Line (428,402) (428,2)
    Meter360 (9,75 196x196), value: MECH.BR.rOUT_PVSpeed, style: Meter-Meter360-Blue, scale format: %d, scale 0..100
    Rectangle (74,219 63x25), "%.1f", text variable: MECH.BR.rOUT_PVSpeed
    Label (465,1 130x20), "Вибратор"
    RockerSwitch (562,56 70x70), variable: MECH.xVibEnable, behaviour: TOGGLE, style: Switch-RockerSwitch-Yellow
    Rectangle (493,65 69x20), "Включен", colour toggle: MECH.xVibEnable
    Rectangle (493,96 69x20), "Отключен", colour toggle: NOT(MECH.xVibEnable)
    Rectangle (446,103 30x25), "%t[ss]", text variable: MECH.VIBRATOR.CLOCK.ET
    Button (494,313 70x70), "ТЕСТ"
        OnMouseDown: execute { MECH.xVibTEST := TRUE; }
        OnMouseUp: execute { MECH.xVibTEST := FALSE; }
    Rectangle (492,25 69x20), "В работе", colour toggle: MECH.Elevator.xOutWork
END_VISUALIZATION

// Device/Application/VMain
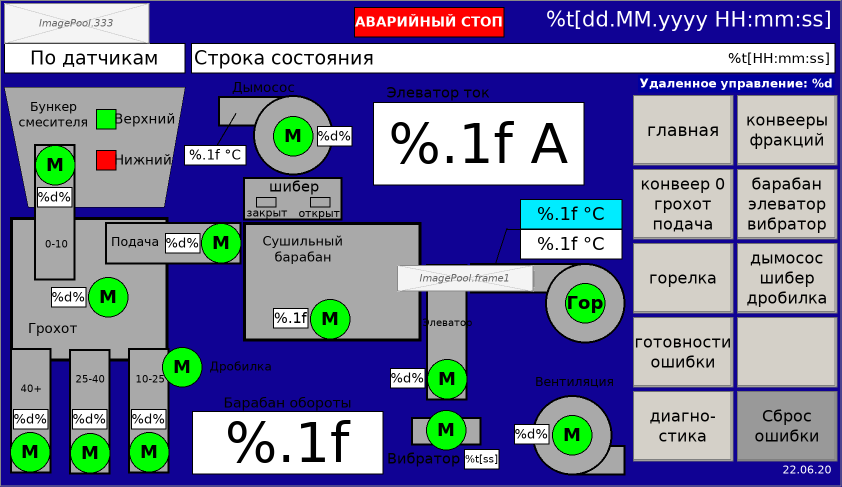
VISUALIZATION VMain  // 842x487
    Frame (-1,79 630x400)
        shows VFr1Main()
        shows VFr2KonvFrak()
        shows VFr3Grohot()
        shows VFr4Baraban()
        shows VFr5Gorelka()
        shows VFr6Dedusting()
        shows VFr7RandE()
        shows VFrADiag()
    Button (633,95 100x70), "главная"
        OnMouseClick: FrameSelectionChange Selection=SelectedFrame=5ddc75d5-edde-4cc6-9f2a-3d195ac39671, GlobSel=AssignType=Directly, SelType=Locally
    Button (737,95 100x70), "конвееры фракций"
        OnMouseClick: FrameSelectionChange Selection=SelectedFrame=5ddc75d5-edde-4cc6-9f2a-3d195ac39671, Selection=1, GlobSel=AssignType=Directly, SelType=Locally
    Button (633,169 100x70), "конвеер 0 грохот подача"
        OnMouseClick: FrameSelectionChange Selection=SelectedFrame=5ddc75d5-edde-4cc6-9f2a-3d195ac39671, Selection=2, GlobSel=AssignType=Directly, SelType=Locally
    Button (737,169 100x70), "барабан элеватор вибратор"
        OnMouseClick: FrameSelectionChange Selection=SelectedFrame=5ddc75d5-edde-4cc6-9f2a-3d195ac39671, Selection=3, GlobSel=AssignType=Directly, SelType=Locally
    Button (633,243 100x70), "горелка"
        OnMouseClick: FrameSelectionChange Selection=SelectedFrame=5ddc75d5-edde-4cc6-9f2a-3d195ac39671, Selection=4, GlobSel=AssignType=Directly, SelType=Locally
    Button (737,243 100x70), "дымосос шибер дробилка"
        OnMouseClick: FrameSelectionChange Selection=SelectedFrame=5ddc75d5-edde-4cc6-9f2a-3d195ac39671, Selection=5, GlobSel=AssignType=Directly, SelType=Locally
    Button (633,317 100x70), "готовности ошибки"
        OnMouseClick: FrameSelectionChange Selection=SelectedFrame=5ddc75d5-edde-4cc6-9f2a-3d195ac39671, Selection=6, GlobSel=AssignType=Directly, SelType=Locally
    Button (737,391 100x70), "Сброс ошибки"
        OnMouseDown: execute { PLC_PRG.xAck := TRUE; }
        OnMouseUp: execute { PLC_PRG.xAck := FALSE; }
    Button (737,317 100x70), input disabled if: TRUE
    Button (633,391 100x70), "диагно- стика"
        OnMouseClick: FrameSelectionChange Selection=SelectedFrame=5ddc75d5-edde-4cc6-9f2a-3d195ac39671, Selection=7, GlobSel=AssignType=Directly, SelType=Locally
    Rectangle (191,43 644x30), "Строка состояния", text list: 'STEPS', text index: Chain.Step
    Rectangle (545,4 288x30), "%t[dd.MM.yyyy HH:mm:ss]"
    Rectangle (4,43 181x30), "По датчикам", text list: 'TextList', text index: 0
    Label (774,455 66x30), "22.06.20"
    Rectangle (728,43 102x30), "%t[HH:mm:ss]", text variable: Chain.TMRWork.ET, invisible if: NOT(MECH.xVibRunAUTO)
    Rectangle (354,7 150x30), "АВАРИЙНЫЙ СТОП", invisible if: PLC_PRG.DInput1.xDI1
    Rectangle (638,75 196x17), "Удаленное управление: %d", text variable: CountWebCli.iCountActivWebVisus, colour toggle: CountWebCli.xAlarm AND PLC_PRG.xFlash
    Image (4,3 145x40), image: ImagePool.333
END_VISUALIZATION

// Device/Application/VFr1Main
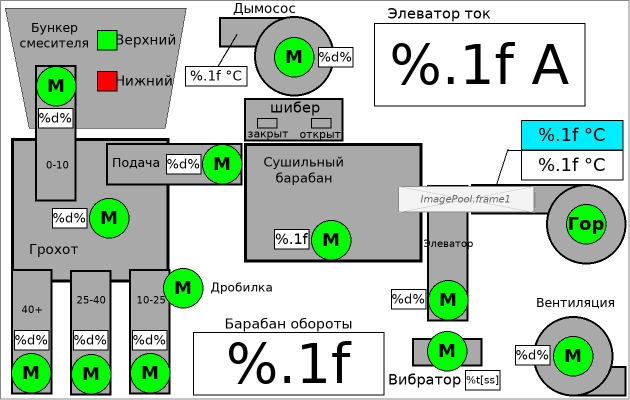
VISUALIZATION VFr1Main  // 630x400, background image ImagePool.fonFreame
    RoundedRectangle (412,338 70x28), colour toggle: MECH.xVibRunAUTO
    RoundedRectangle (11,138 158x144)
    Polygon (5,8) (79,8) (186,8) (165,128) (29,128)
    RoundedRectangle (129,269 41x125)
    RoundedRectangle (70,270 41x125)
    RoundedRectangle (11,269 41x125)
    RoundedRectangle (35,65 41x136)
    Ellipse (36,66 40x40), "М", colour toggle: MECH.K0.xOUT_Error
    Ellipse (11,353 40x40), "М", colour toggle: MECH.K40.xOUT_Error
    Ellipse (71,354 40x40), "М", colour toggle: MECH.K25.xOUT_Error
    Ellipse (130,353 40x40), "М", colour toggle: MECH.K10.xOUT_Error
    Ellipse (89,198 40x40), "М", colour toggle: MECH.Gr.xOUT_Error
    Rectangle (97,30 20x20), colour toggle: PLC_PRG.DInput1.xDI2
    Label (114,30 64x20), "Верхний"
    Rectangle (97,71 20x20), colour toggle: PLC_PRG.DInput1.xDI3
    Label (112,71 64x20), "Нижний"
    Rectangle (244,143 178x119)
    Ellipse (311,220 40x40), "М", colour toggle: MECH.BR.xOUT_Error
    Rectangle (244,98 99x43)
    Label (289,125 63x19), "открыт"
    Rectangle (311,118 20x10), colour toggle: PLC_PRG.DInput2.xDI1
    Label (236,124 64x20), "закрыт"
    Rectangle (257,118 20x10), colour toggle: PLC_PRG.DInput2.xDI2
    Rectangle (219,17 78x30)
    Ellipse (254,16 80x80)
    Ellipse (274,37 40x40), "М", colour toggle: MECH.Ded.xOUT_Error
    Rectangle (471,184 118x30)
    Ellipse (546,184 80x80)
    Ellipse (566,204 40x40), "Гор"
    Rectangle (571,366 55x30)
    Ellipse (533,316 80x80)
    Ellipse (553,336 40x40), "М"
    RoundedRectangle (427,185 41x136)
    Ellipse (428,280 40x40), "М", colour toggle: MECH.EL.xOUT_Error
    Ellipse (427,331 40x40), "М"
    Group (496,149 25x50)
        Line (0,37) (12,0)
        Line (12,1) (25,1)
    RoundedRectangle (185,66 62x20), "%.1f °C", text variable: MECH.rOutDedPVTemp
    Rectangle (521,150 102x30), "%.1f °C", text variable: MECH.rOutGorPVTemp
    Rectangle (521,120 102x30), "%.1f °C", text variable: MECH.rOutGorSPTemp
    Ellipse (36,66 40x40), "М", invisible if: NOT(MECH.K0.xOUT_Work)
    Ellipse (11,353 40x40), "М", invisible if: NOT(MECH.K40.xOUT_Work)
    Ellipse (71,354 40x40), "М", invisible if: NOT(MECH.K25.xOUT_Work)
    Ellipse (130,353 40x40), "М", invisible if: NOT(MECH.K10.xOUT_Work)
    Ellipse (89,198 40x40), "М", invisible if: NOT(MECH.Gr.xOUT_Work)
    Ellipse (311,220 40x40), "М", invisible if: NOT(MECH.BR.xOUT_Work)
    Ellipse (274,37 40x40), "М", invisible if: NOT(MECH.Ded.xOUT_Work)
    Ellipse (566,204 40x40), "Гор", invisible if: NOT(MECH.xGorRun)
    Ellipse (428,280 40x40), "М", invisible if: NOT(MECH.EL.xOUT_Work)
    Ellipse (427,331 40x40), "М", invisible if: NOT(MECH.xVibRun)
    RoundedRectangle (106,143 136x42)
    Ellipse (202,144 40x40), "М", colour toggle: MECH.PD.xOUT_Error
    Ellipse (202,144 40x40), "М", invisible if: NOT(MECH.PD.xOUT_Work)
    RoundedRectangle (15,300 35x21), angle 270, "40+"
    RoundedRectangle (65,290 52x21), angle 270, "25-40"
    RoundedRectangle (125,290 52x21), angle 270, "10-25"
    RoundedRectangle (31,155 52x21), angle 270, "0-10"
    RoundedRectangle (28,239 52x21), "Грохот"
    RoundedRectangle (18,16 73x39), "Бункер смесителя"
    RoundedRectangle (110,152 52x21), "Подача"
    RoundedRectangle (263,152 82x36), "Сушильный барабан"
    RoundedRectangle (269,97 52x21), "шибер"
    RoundedRectangle (232,-2 65x21), "Дымосос"
    RoundedRectangle (412,234 73x21), angle 270, "Элеватор"
    RoundedRectangle (387,369 75x21), "Вибратор"
    RoundedRectangle (534,292 83x21), "Вентиляция"
    RoundedRectangle (14,330 35x20), "%d%", text variable: MECH.K40.iOUT_PVSpeed
    RoundedRectangle (73,330 35x20), "%d%", text variable: MECH.K25.iOUT_PVSpeed
    RoundedRectangle (132,330 35x20), "%d%", text variable: MECH.K25.iOUT_PVSpeed
    RoundedRectangle (52,208 35x20), "%d%", text variable: MECH.Gr.iOUT_PVSpeed
    RoundedRectangle (38,108 35x20), "%d%", text variable: MECH.K0.iOUT_PVSpeed
    RoundedRectangle (166,154 35x20), "%d%", text variable: MECH.PD.iOUT_PVSpeed
    RoundedRectangle (318,47 35x20), "%d%", text variable: MECH.Ded.iOUT_PVSpeed
    RoundedRectangle (274,229 35x20), "%.1f", text variable: MECH.BR.rOUT_PVSpeed
    RoundedRectangle (391,289 35x20), "%d%", text variable: MECH.EL.iOUT_PVSpeed
    Line (218,66) (237,34)
    RoundedRectangle (374,23 211x83), "%.1f A", text variable: MECH.EL.rOUT_Current
    RoundedRectangle (193,332 191x63), "%.1f", text variable: MECH.BR.rOUT_PVSpeed
    RoundedRectangle (223,313 131x21), "Барабан обороты"
    Ellipse (553,336 40x40), "М", invisible if: NOT(MECH.xVentWork)
    RoundedRectangle (515,345 35x20), "%d%", text variable: MECH.rOutVentPVSpeed
    RoundedRectangle (465,370 35x20), "%t[ss]", text variable: MECH.VIBRATOR.CLOCK.ET
    RoundedRectangle (386,3 107x21), "Элеватор ток"
    Ellipse (163,268 40x40), "М", colour toggle: MECH.xDrob_OUT_Error
    Ellipse (163,268 40x40), "М", invisible if: NOT(MECH.xDrob_OUT_Work)
    RoundedRectangle (209,277 66x21), "Дробилка"
    Image (479,191 56x17), invisible if: NOT(MECH.xGorNagrevONOFF AND MECH.xGorWork), image: ImagePool.frame1
    Line (534,214) (534,184)
    Image (398,186 136x26), invisible if: NOT(MECH.xGorNagrevONOFF AND MECH.xGor2Stup AND MECH.xGorWork), image: ImagePool.frame1
END_VISUALIZATION

// Device/Application/VFr2KonvFrak
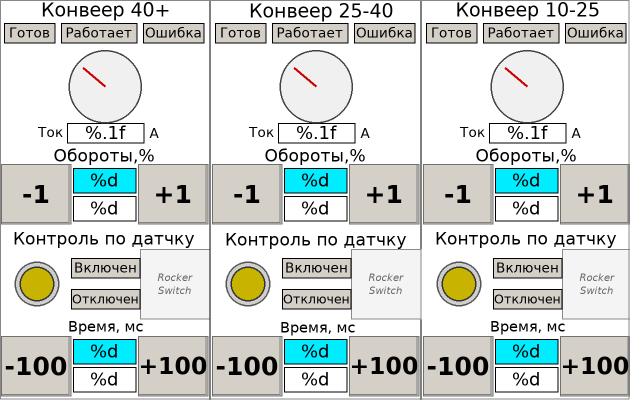
VISUALIZATION VFr2KonvFrak  // 630x400, background image ImagePool.fonFreame
    Rectangle (73,196 63x25), "%d", text variable: MECH.K40.iOUT_PVSpeed
    Rectangle (73,168 63x25), "%d", text variable: MECH.K40_iIN_SPSpeed
    Button (138,164 70x60), "+1"
        OnMouseClick: execute {
            IF MECH.K40_iIN_SPSpeed <100 THEN
            	MECH.K40_iIN_SPSpeed := MECH.K40_iIN_SPSpeed + 1;
            END_IF;
        }
    Button (1,164 70x60), "-1"
        OnMouseClick: execute {
            IF MECH.K40_iIN_SPSpeed >5 THEN
            	MECH.K40_iIN_SPSpeed := MECH.K40_iIN_SPSpeed - 1;
            END_IF;
        }
    Label (41,0 130x20), "Конвеер 40+"
    Rectangle (67,123 77x20), "%.1f", text variable: MECH.K40.rOUT_Current
    Label (22,123 57x19), "Ток"
    Label (57,148 94x15), "Обороты,%"
    Rectangle (73,367 63x25), "%d", text variable: MECH.K40.iOUT_PVRotation, colour toggle: MECH.Konveer40.xFirstRun
    Rectangle (73,339 63x25), "%d", text variable: MECH.K40_iIN_SPRotatTimeMS
    Button (138,336 70x60), "+100"
        OnMouseClick: execute {
            IF MECH.K40_iIN_SPRotatTimeMS <10000 THEN
            	MECH.K40_iIN_SPRotatTimeMS := MECH.K40_iIN_SPRotatTimeMS + 100;
            END_IF;
        }
    Button (1,336 70x60), "-100"
        OnMouseClick: execute {
            IF MECH.K40_iIN_SPRotatTimeMS >500 THEN
            	MECH.K40_iIN_SPRotatTimeMS := MECH.K40_iIN_SPRotatTimeMS - 100;
            END_IF;
        }
    Label (2,229 204x19), "Контроль по датчку"
    RockerSwitch (140,249 70x70), variable: MECH.K40_xIN_EnCtrlSensor, behaviour: TOGGLE, style: Switch-RockerSwitch-Yellow
    Meter180 (33,50 144x73), value: MECH.K40.rOUT_Current, style: Meter-Meter180-Green, scale format: %d, scale 0..10
    Line (210,400) (210,0)
    Line (421,400) (421,0)
    Rectangle (61,23 76x20), "Работает", colour toggle: MECH.K40.xOUT_Work
    Rectangle (143,23 61x20), "Ошибка", colour toggle: MECH.K40.xOUT_Error
    Rectangle (4,23 51x20), "Готов", colour toggle: MECH.K40.xOUT_Ready
    Label (139,124 30x19), "А"
    Lamp1 (10,258 54x52), variable: PLC_PRG.DInput1.xDI15, style: Lamp-Lamp1-Yellow
    Label (4,317 204x19), "Время, мс"
    Rectangle (71,258 69x20), "Включен", colour toggle: MECH.K40_xIN_EnCtrlSensor
    Rectangle (71,289 69x20), "Отключен", colour toggle: NOT(MECH.K40_xIN_EnCtrlSensor)
    Rectangle (284,196 63x25), "%d", text variable: MECH.K25.iOUT_PVSpeed
    Rectangle (284,168 63x25), "%d", text variable: MECH.K25_iIN_SPSpeed
    Button (349,164 70x60), "+1"
        OnMouseClick: execute {
            IF MECH.K25_iIN_SPSpeed <100 THEN
            	MECH.K25_iIN_SPSpeed := MECH.K25_iIN_SPSpeed + 1;
            END_IF;
        }
    Button (212,164 70x60), "-1"
        OnMouseClick: execute {
            IF MECH.K25_iIN_SPSpeed >5 THEN
            	MECH.K25_iIN_SPSpeed := MECH.K25_iIN_SPSpeed - 1;
            END_IF;
        }
    Label (249,1 145x20), "Конвеер 25-40"
    Rectangle (278,123 77x20), "%.1f", text variable: MECH.K25.rOUT_Current
    Label (233,123 57x19), "Ток"
    Label (268,148 94x15), "Обороты,%"
    Rectangle (284,367 63x25), "%d", text variable: MECH.K25.iOUT_PVRotation, colour toggle: MECH.Konveer25.xFirstRun
    Rectangle (284,339 63x25), "%d", text variable: MECH.K25_iIN_SPRotatTimeMS
    Button (349,336 70x60), "+100"
        OnMouseClick: execute {
            IF MECH.K25_iIN_SPRotatTimeMS <10000 THEN
            	MECH.K25_iIN_SPRotatTimeMS := MECH.K25_iIN_SPRotatTimeMS + 100;
            END_IF;
        }
    Button (212,336 70x60), "-100"
        OnMouseClick: execute {
            IF MECH.K25_iIN_SPRotatTimeMS >500 THEN
            	MECH.K25_iIN_SPRotatTimeMS := MECH.K25_iIN_SPRotatTimeMS - 100;
            END_IF;
        }
    RockerSwitch (351,249 70x70), variable: MECH.K25_xIN_EnCtrlSensor, behaviour: TOGGLE, style: Switch-RockerSwitch-Yellow
    Meter180 (244,50 144x73), value: MECH.K25.rOUT_Current, style: Meter-Meter180-Green, scale format: %d, scale 0..10
    Rectangle (272,23 76x20), "Работает", colour toggle: MECH.K25.xOUT_Work
    Rectangle (354,23 61x20), "Ошибка", colour toggle: MECH.K25.xOUT_Error
    Rectangle (215,23 51x20), "Готов", colour toggle: MECH.K25.xOUT_Ready
    Label (350,124 30x19), "А"
    Lamp1 (221,258 54x52), variable: PLC_PRG.DInput1.xDI16, style: Lamp-Lamp1-Yellow
    Rectangle (282,258 69x20), "Включен", colour toggle: MECH.K25_xIN_EnCtrlSensor
    Rectangle (282,289 69x20), "Отключен", colour toggle: NOT(MECH.K25_xIN_EnCtrlSensor)
    Rectangle (495,196 63x25), "%d", text variable: MECH.K10.iOUT_PVSpeed
    Rectangle (495,168 63x25), "%d", text variable: MECH.K10_iIN_SPSpeed
    Button (560,164 70x60), "+1"
        OnMouseClick: execute {
            IF MECH.K10_iIN_SPSpeed <100 THEN
            	MECH.K10_iIN_SPSpeed := MECH.K10_iIN_SPSpeed + 1;
            END_IF;
        }
    Button (423,164 70x60), "-1"
        OnMouseClick: execute {
            IF MECH.K10_iIN_SPSpeed >5 THEN
            	MECH.K10_iIN_SPSpeed := MECH.K10_iIN_SPSpeed - 1;
            END_IF;
        }
    Label (453,0 150x20), "Конвеер 10-25"
    Rectangle (489,123 77x20), "%.1f", text variable: MECH.K10.rOUT_Current
    Label (444,123 57x19), "Ток"
    Label (479,148 94x15), "Обороты,%"
    Rectangle (495,367 63x25), "%d", text variable: MECH.K10.iOUT_PVRotation, colour toggle: MECH.Konveer10.xFirstRun
    Rectangle (495,339 63x25), "%d", text variable: MECH.K10_iIN_SPRotatTimeMS
    Button (560,336 70x60), "+100"
        OnMouseClick: execute {
            IF MECH.K10_iIN_SPRotatTimeMS <10000 THEN
            	MECH.K10_iIN_SPRotatTimeMS := MECH.K10_iIN_SPRotatTimeMS + 100;
            END_IF;
        }
    Button (423,336 70x60), "-100"
        OnMouseClick: execute {
            IF MECH.K10_iIN_SPRotatTimeMS >500 THEN
            	MECH.K10_iIN_SPRotatTimeMS := MECH.K10_iIN_SPRotatTimeMS - 100;
            END_IF;
        }
    RockerSwitch (562,249 70x70), variable: MECH.K10_xIN_EnCtrlSensor, behaviour: TOGGLE, style: Switch-RockerSwitch-Yellow
    Meter180 (455,50 144x73), value: MECH.K10.rOUT_Current, style: Meter-Meter180-Green, scale format: %d, scale 0..10
    Rectangle (483,23 76x20), "Работает", colour toggle: MECH.K10.xOUT_Work
    Rectangle (565,23 61x20), "Ошибка", colour toggle: MECH.K10.xOUT_Error
    Rectangle (426,23 51x20), "Готов", colour toggle: MECH.K10.xOUT_Ready
    Label (561,124 30x19), "А"
    Lamp1 (432,258 54x52), variable: PLC_PRG.DInput1.xDI17, style: Lamp-Lamp1-Yellow
    Rectangle (493,258 69x20), "Включен", colour toggle: MECH.K10_xIN_EnCtrlSensor
    Rectangle (493,289 69x20), "Отключен", colour toggle: NOT(MECH.K10_xIN_EnCtrlSensor)
    Label (216,318 204x19), "Время, мс"
    Label (214,230 204x19), "Контроль по датчку"
    Label (426,317 204x19), "Время, мс"
    Label (424,229 204x19), "Контроль по датчку"
END_VISUALIZATION

// Device/Application/VFr3Grohot
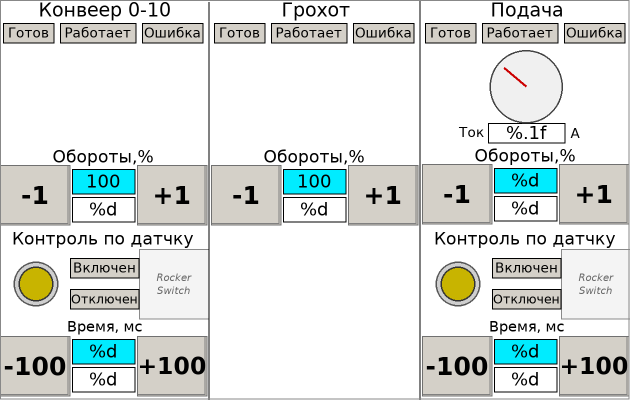
VISUALIZATION VFr3Grohot  // 630x400, background image ImagePool.fonFreame
    Label (40,0 130x20), "Конвеер 0-10"
    Rectangle (72,367 63x25), "%d", text variable: MECH.K0.iOUT_PVRotation, colour toggle: MECH.Konveer0.xFirstRun
    Rectangle (72,339 63x25), "%d", text variable: MECH.K0_iIN_SPRotatTimeMS
    Button (137,336 70x60), "+100"
        OnMouseClick: execute {
            IF MECH.K0_iIN_SPRotatTimeMS <10000 THEN
            	MECH.K0_iIN_SPRotatTimeMS := MECH.K0_iIN_SPRotatTimeMS + 100;
            END_IF;
        }
    Label (1,229 204x19), "Контроль по датчку"
    RockerSwitch (139,249 70x70), variable: MECH.K0_xIN_EnCtrlSensor, behaviour: TOGGLE, style: Switch-RockerSwitch-Yellow
    Rectangle (60,23 76x20), "Работает", colour toggle: MECH.K0.xOUT_Work
    Rectangle (142,23 61x20), "Ошибка", colour toggle: MECH.K0.xOUT_Error
    Rectangle (3,23 51x20), "Готов", colour toggle: MECH.K0.xOUT_Ready
    Lamp1 (9,258 54x52), variable: PLC_PRG.DInput1.xDI18, style: Lamp-Lamp1-Yellow
    Label (3,317 204x19), "Время, мс"
    Rectangle (70,258 69x20), "Включен", colour toggle: MECH.K0_xIN_EnCtrlSensor
    Rectangle (70,289 69x20), "Отключен", colour toggle: NOT(MECH.K0_xIN_EnCtrlSensor)
    Label (251,0 130x20), "Грохот"
    Rectangle (271,23 76x20), "Работает", colour toggle: MECH.Gr.xOUT_Work
    Rectangle (353,23 61x20), "Ошибка", colour toggle: MECH.Gr.xOUT_Error
    Rectangle (214,23 51x20), "Готов", colour toggle: MECH.Gr.xOUT_Ready
    Rectangle (494,196 63x25), "%d", text variable: MECH.PD.iOUT_PVSpeed
    Rectangle (494,168 63x25), "%d", text variable: MECH.iSP_Podacha
    Button (559,164 70x60), "+1", invisible if: TRUE
        OnMouseClick: execute {
            IF MECH.PD_iIN_SPSpeed <100 THEN
            	MECH.PD_iIN_SPSpeed := MECH.PD_iIN_SPSpeed + 1;
            END_IF;
        }
    Button (422,164 70x60), "-1", invisible if: TRUE
        OnMouseClick: execute {
            IF MECH.PD_iIN_SPSpeed >5 THEN
            	MECH.PD_iIN_SPSpeed := MECH.PD_iIN_SPSpeed - 1;
            END_IF;
        }
    Label (462,0 130x20), "Подача"
    Rectangle (488,123 77x20), "%.1f", text variable: MECH.PD.rOUT_Current
    Label (443,123 57x19), "Ток"
    Label (478,148 94x15), "Обороты,%"
    Rectangle (494,367 63x25), "%d", text variable: MECH.PD.iOUT_PVRotation, colour toggle: MECH.Podacha.xFirstRun
    Rectangle (494,339 63x25), "%d", text variable: MECH.PD_iIN_SPRotatTimeMS
    Button (559,336 70x60), "+100"
        OnMouseClick: execute {
            IF MECH.PD_iIN_SPRotatTimeMS <10000 THEN
            	MECH.PD_iIN_SPRotatTimeMS := MECH.PD_iIN_SPRotatTimeMS + 100;
            END_IF;
        }
    Button (422,336 70x60), "-100"
        OnMouseClick: execute {
            IF MECH.PD_iIN_SPRotatTimeMS >500 THEN
            	MECH.PD_iIN_SPRotatTimeMS := MECH.PD_iIN_SPRotatTimeMS - 100;
            END_IF;
        }
    RockerSwitch (561,249 70x70), variable: MECH.PD_xIN_EnCtrlSensor, behaviour: TOGGLE, style: Switch-RockerSwitch-Yellow
    Meter180 (454,50 144x73), value: MECH.PD.rOUT_Current, style: Meter-Meter180-Green, scale format: %d, scale 0..10
    Rectangle (482,23 76x20), "Работает", colour toggle: MECH.PD.xOUT_Work
    Rectangle (564,23 61x20), "Ошибка", colour toggle: MECH.PD.xOUT_Error
    Rectangle (425,23 51x20), "Готов", colour toggle: MECH.PD.xOUT_Ready
    Label (560,124 30x19), "А"
    Lamp1 (431,258 54x52), variable: PLC_PRG.DInput1.xDI19, style: Lamp-Lamp1-Yellow
    Rectangle (492,258 69x20), "Включен", colour toggle: MECH.PD_xIN_EnCtrlSensor
    Rectangle (492,289 69x20), "Отключен", colour toggle: NOT(MECH.PD_xIN_EnCtrlSensor)
    Label (425,317 204x19), "Время, мс"
    Label (423,229 204x19), "Контроль по датчку"
    Button (0,336 70x60), "-100"
        OnMouseClick: execute {
            IF MECH.K0_iIN_SPRotatTimeMS >500 THEN
            	MECH.K0_iIN_SPRotatTimeMS := MECH.K0_iIN_SPRotatTimeMS - 100;
            END_IF;
        }
    Line (209,402) (209,2)
    Line (420,400) (420,0)
    Button (211,165 70x60), "-1", input disabled if: TRUE
    Rectangle (283,197 63x25), "%d", text variable: MECH.Grohot.iOutPVSpeed
    Rectangle (283,169 63x25), "100"
    Button (348,165 70x60), "+1", input disabled if: TRUE
    Label (267,149 94x15), "Обороты,%"
    Button (0,165 70x60), "-1", input disabled if: TRUE
    Rectangle (72,197 63x25), "%d", text variable: MECH.Konveer0.iOutPVSpeed
    Rectangle (72,169 63x25), "100"
    Button (137,165 70x60), "+1", input disabled if: TRUE
    Label (56,149 94x15), "Обороты,%"
END_VISUALIZATION

// Device/Application/VFr5Gorelka
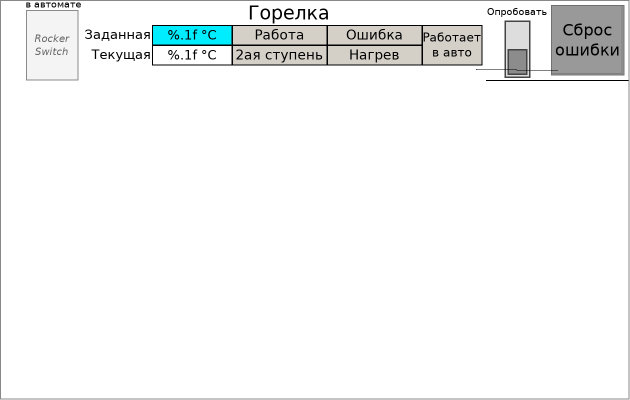
VISUALIZATION VFr5Gorelka  // 630x400, background image ImagePool.fonFreame
    Rectangle (152,25 80x20), "%.1f °C", text variable: MECH.rOutGorSPTemp
    Rectangle (152,45 80x20), "%.1f °C", text variable: MECH.rOutGorPVTemp
    Rectangle (327,25 95x20), "Ошибка", colour toggle: MECH.xGorFaultRS.Q1
    Label (224,3 130x20), "Горелка"
    Rectangle (232,25 95x20), "Работа", colour toggle: MECH.xGorWork
    Rectangle (232,45 95x20), "2ая ступень", colour toggle: MECH.xGor2Stup
    Rectangle (422,25 60x40), "Работает в авто", colour toggle: MECH.xGorRunAUTO
    RockerSwitch (26,10 52x70), variable: MECH.xGorSwitchRun, behaviour: TOGGLE, style: Switch-RockerSwitch-Green
    Label (8,-2 91x13), "в автомате"
    Label (92,23 62x23), "Заданная"
    Label (96,43 58x23), "Текущая"
    Label (477,1 80x22), "Опробовать"
    DipSwitch (489,20 57x58), variable: MECH.xGorOprob, input disabled if: MECH.K40.xIN_Run OR NOT(PLC_PRG.DInput1.xDI1), behaviour: TOGGLE, style: Switch-DipSwitch-Gray
    Button (551,5 73x70), "Сброс ошибки"
        OnMouseDown: execute { MECH.xGorAckButton := TRUE; }
        OnMouseUp: execute { MECH.xGorAckButton := FALSE; }
    Rectangle (327,45 95x20), "Нагрев", colour toggle: MECH.xGorNagrevONOFF
    Line (486,80) (629,80)
    Line (476,69) (557,70)
END_VISUALIZATION

// Device/Application/VFr6Dedusting
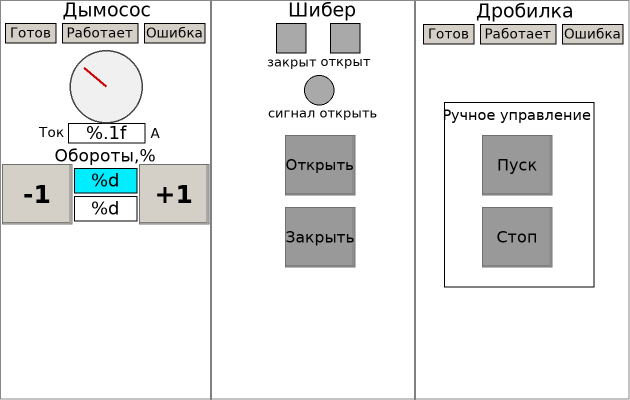
VISUALIZATION VFr6Dedusting  // 630x400, background image ImagePool.fonFreame
    Rectangle (444,102 150x185)
    Rectangle (74,196 63x25), "%d", text variable: MECH.Ded.iOUT_PVSpeed
    Rectangle (74,168 63x25), "%d", text variable: MECH.Ded_iIN_SPSpeed
    Button (139,164 70x60), "+1"
        OnMouseClick: execute {
            IF MECH.Ded_iIN_SPSpeed <100 THEN
            	MECH.Ded_iIN_SPSpeed := MECH.Ded_iIN_SPSpeed + 1;
            END_IF;
        }
    Button (2,164 70x60), "-1"
        OnMouseClick: execute {
            IF MECH.Ded_iIN_SPSpeed >5 THEN
            	MECH.Ded_iIN_SPSpeed := MECH.Ded_iIN_SPSpeed - 1;
            END_IF;
        }
    Label (42,0 130x20), "Дымосос"
    Rectangle (68,123 77x20), "%.1f", text variable: MECH.Ded.rOUT_Current
    Label (23,123 57x19), "Ток"
    Label (58,148 94x15), "Обороты,%"
    Meter180 (34,50 144x73), value: MECH.Ded.rOUT_Current, style: Meter-Meter180-Green, scale format: %d, scale 0..10
    Rectangle (62,23 76x20), "Работает", colour toggle: MECH.Ded.xOUT_Work
    Rectangle (144,23 61x20), "Ошибка", colour toggle: MECH.Ded.xOUT_Error
    Rectangle (5,23 51x20), "Готов", colour toggle: MECH.Ded.xOUT_Ready
    Label (140,124 30x19), "А"
    Line (211,401) (211,1)
    Label (257,0 130x20), "Шибер"
    Button (285,135 70x60), "Открыть", input disabled if: MECH.Ded.xOUT_Work
        OnMouseDown: execute { PLC_PRG.DOutput1.xDO12 := TRUE; }
    Button (285,207 70x60), "Закрыть", input disabled if: MECH.Ded.xOUT_Work
        OnMouseDown: execute { PLC_PRG.DOutput1.xDO12 := FALSE; }
    Rectangle (330,23 30x30), colour toggle: PLC_PRG.DInput2.xDI1
    Label (314,52 63x19), "открыт"
    Label (260,52 64x20), "закрыт"
    Rectangle (276,23 30x30), colour toggle: PLC_PRG.DInput2.xDI2
    Label (267,103 111x20), "сигнал открыть"
    Ellipse (304,75 30x30), colour toggle: PLC_PRG.DOutput1.xDO12
    Line (415,400) (415,0)
    Label (460,1 130x20), "Дробилка"
    Rectangle (480,24 76x20), "Работает", colour toggle: MECH.xDrob_OUT_Work
    Rectangle (562,24 61x20), "Ошибка", colour toggle: MECH.xDrob_OUT_Error
    Rectangle (423,24 51x20), "Готов", colour toggle: MECH.xDrob_OUT_Ready
    Button (482,207 70x60), "Стоп", invisible if: Chain.xLampPUSK, input disabled if: Chain.xLampPUSK
        OnMouseDown: execute { MECH.xDrobRun := FALSE; }
    Button (482,135 70x60), "Пуск", invisible if: Chain.xLampPUSK, input disabled if: Chain.xLampPUSK
        OnMouseDown: execute { MECH.xDrobRun := TRUE; }
    Label (452,105 130x20), "Ручное управление"
END_VISUALIZATION

// Device/Application/VFr7RandE
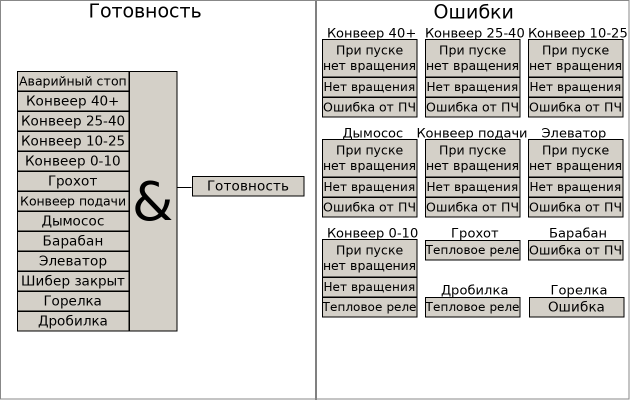
VISUALIZATION VFr7RandE  // 630x400, background image ImagePool.fonFreame
    Label (409,2 130x20), "Ошибки"
    Label (80,1 130x20), "Готовность"
    Line (316,401) (316,1)
    Rectangle (322,39 95x38), "При пуске нет вращения", colour toggle: MECH.Konveer40.xStartNoRotation
    Rectangle (17,71 112x20), "Аварийный стоп", colour toggle: PLC_PRG.DInput1.xDI1
    Rectangle (17,91 112x20), "Конвеер 40+", colour toggle: MECH.K40.xOUT_Ready
    Rectangle (17,111 112x20), "Конвеер 25-40", colour toggle: MECH.K25.xOUT_Ready
    Rectangle (17,131 112x20), "Конвеер 10-25", colour toggle: MECH.K10.xOUT_Ready
    Rectangle (17,151 112x20), "Конвеер 0-10", colour toggle: MECH.K0.xOUT_Ready
    Rectangle (17,171 112x20), "Грохот", colour toggle: MECH.Gr.xOUT_Ready
    Rectangle (17,191 112x20), "Конвеер подачи", colour toggle: MECH.PD.xOUT_Ready
    Rectangle (17,211 112x20), "Дымосос", colour toggle: MECH.Ded.xOUT_Ready
    Rectangle (17,231 112x20), "Барабан", colour toggle: MECH.BR.xOUT_Ready
    Rectangle (17,251 112x20), "Элеватор", colour toggle: MECH.EL.xOUT_Ready
    Rectangle (17,271 112x20), "Шибер закрыт", colour toggle: PLC_PRG.DInput2.xDI2
    Rectangle (17,291 112x20), "Горелка", colour toggle: NOT(MECH.xGorOprob)
    Rectangle (129,71 48x260), "&", colour toggle: Chain.ReadyRun
    Rectangle (192,176 112x20), "Готовность", colour toggle: Chain.ReadyRun
    Line (177,187) (191,187)
    Label (307,23 130x20), "Конвеер 40+"
    Rectangle (322,77 95x20), "Нет вращения", colour toggle: MECH.Konveer40.xNoRation
    Rectangle (322,97 95x20), "Ошибка от ПЧ", colour toggle: MECH.Konveer40.xExtError
    Rectangle (425,39 95x38), "При пуске нет вращения", colour toggle: MECH.Konveer25.xStartNoRotation
    Label (410,23 130x20), "Конвеер 25-40"
    Rectangle (425,77 95x20), "Нет вращения", colour toggle: MECH.Konveer25.xNoRation
    Rectangle (425,97 95x20), "Ошибка от ПЧ", colour toggle: MECH.Konveer25.xExtError
    Rectangle (528,39 95x38), "При пуске нет вращения", colour toggle: MECH.Konveer10.xStartNoRotation
    Label (513,23 130x20), "Конвеер 10-25"
    Rectangle (528,77 95x20), "Нет вращения", colour toggle: MECH.Konveer10.xNoRation
    Rectangle (528,97 95x20), "Ошибка от ПЧ", colour toggle: MECH.Konveer10.xExtError
    Rectangle (322,139 95x38), "При пуске нет вращения", colour toggle: MECH.Dedusting.xStartNoRotation
    Label (308,223 130x20), "Конвеер 0-10"
    Rectangle (322,177 95x20), "Нет вращения", colour toggle: MECH.Dedusting.xNoRation
    Rectangle (322,197 95x20), "Ошибка от ПЧ", colour toggle: MECH.Dedusting.xExtError
    Rectangle (425,139 95x38), "При пуске нет вращения", colour toggle: MECH.Podacha.xStartNoRotation
    Label (407,123 130x20), "Конвеер подачи"
    Rectangle (425,177 95x20), "Нет вращения", colour toggle: MECH.Podacha.xNoRation
    Rectangle (425,197 95x20), "Ошибка от ПЧ", colour toggle: MECH.Podacha.xExtError
    Rectangle (528,139 95x38), "При пуске нет вращения", colour toggle: MECH.Elevator.xStartNoRotation
    Label (308,123 130x20), "Дымосос"
    Rectangle (528,177 95x20), "Нет вращения", colour toggle: MECH.Elevator.xNoRation
    Rectangle (528,197 95x20), "Ошибка от ПЧ", colour toggle: MECH.Elevator.xExtError
    Rectangle (322,239 95x38), "При пуске нет вращения", colour toggle: MECH.Konveer0.xStartNoRotation
    Label (509,123 130x20), "Элеватор"
    Rectangle (322,277 95x20), "Нет вращения", colour toggle: MECH.Konveer0.xNoRation
    Rectangle (322,297 95x20), "Тепловое реле", colour toggle: MECH.Konveer0.xExtError
    Label (410,223 130x20), "Грохот"
    Rectangle (425,240 95x20), "Тепловое реле", colour toggle: MECH.Grohot.xExtError
    Label (513,223 130x20), "Барабан"
    Rectangle (528,240 95x20), "Ошибка от ПЧ", colour toggle: MECH.Baraban.xExtError
    Rectangle (529,297 95x20), "Ошибка", colour toggle: MECH.xGorFaultRS.Q1
    Label (514,280 130x20), "Горелка"
    Rectangle (425,297 95x20), "Тепловое реле", colour toggle: MECH.xDrob_OUT_Error
    Label (410,280 130x20), "Дробилка"
    Rectangle (17,311 112x20), "Дробилка", colour toggle: MECH.xDrob_OUT_Ready
END_VISUALIZATION

(* text list TextList (id | default)
  0 | Первый
  1 | Второй
  2 | Третий
  3 | Четвертый
   |  *)

(* text list System (id | default)
  Apr | Apr
  April | April
  Aug | Aug
  August | August
  Dec | Dec
  December | December
  Feb | Feb
  February | February
  Fri | Fri
  Friday | Friday
  Jan | Jan
  January | January
  Jul | Jul
  July | July
  Jun | Jun
  June | June
  Mar | Mar
  March | March
  May | May
  May_3Letter | May
  Mon | Mon
  Monday | Monday
  Nov | Nov
  November | November
  Oct | Oct
  October | October
  Sat | Sat
  Saturday | Saturday
  Sep | Sep
  September | September
  Sun | Sun
  Sunday | Sunday
  Thu | Thu
  Thursday | Thursday
  Tue | Tue
  Tuesday | Tuesday
  Wed | Wed
  Wednesday | Wednesday
   |  *)

(* text list STEPS (id | default)
  0 | ГОТОВ
  1 | НЕТ ГОТОВНОСТИ
  5 | Запуск К40, К25, К10, К0, дымососа
  995 | Останов К40, К25, К10, К0, дымососа
  1000 | АВАРИЙНЫЙ СТОП
  10 | Запуск грохота
  15 | Запуск подающего конвеера
  990 | Останов грохота
  985 | Останов подающего конвеера
  20 | Запуск барабана и горелки
  25 | Запуск элеватора
  30 | Работа                                                        Время работы:
  970 | Остановка вибратора
  975 | Остановка элеватора
  980 | Остановка барабана и горелки
   |  *)
